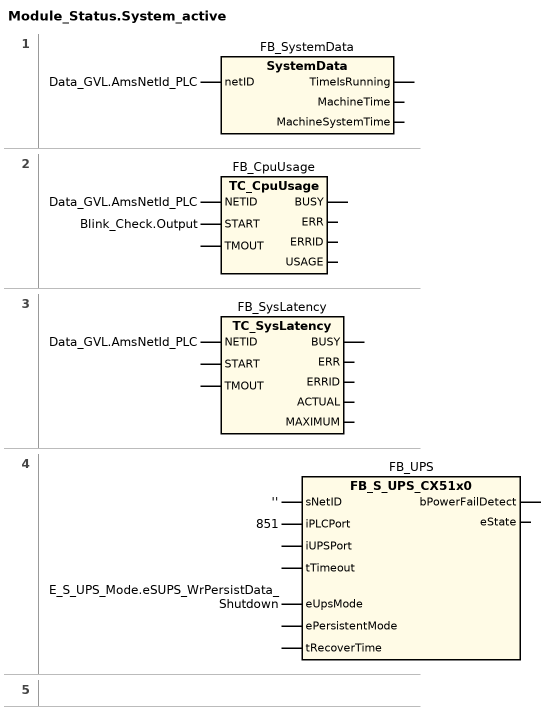
// NETWORK 1
FB_SystemData(netID := Data_GVL.AmsNetId_PLC); // SystemData

// NETWORK 2
FB_CpuUsage(NETID := Data_GVL.AmsNetId_PLC, START := Blink_Check.Output); // TC_CpuUsage

// NETWORK 3
FB_SysLatency(NETID := Data_GVL.AmsNetId_PLC); // TC_SysLatency

// NETWORK 4
FB_UPS(sNetID := '', iPLCPort := 851, eUpsMode := E_S_UPS_Mode.eSUPS_WrPersistData_Shutdown); // FB_S_UPS_CX51x0

// NETWORK 5
END_ACTION

END_PROGRAM

// ---- POUs/Function_Block/General/Ethercat_Status.TcPOU
FUNCTION_BLOCK Ethercat_Status
VAR_IN_OUT 
	stSlaveCurrentState			: stEcSlaveState;
END_VAR
VAR_INPUT
   bEnable: BOOL;                                               (*Enabling FB on rising edge*)
   sNetId: STRING;                                              (*Master's EtherCAT NetId*)
   nSlaveAddr: UINT;                                            (*Slave's EtherCAT address*)
END_VAR
VAR_OUTPUT
   bDone: BOOL;                                                 (*Successfully done*)
   iMessage: STRING (10);                                       (*String message*)
   bError: BOOL;                                                (*Error detected*)
   nErrId: UDINT;                                               (*ADS error code*)
   stActualState: ST_EcSlaveState;                              (*Actual slave status*)
END_VAR
VAR
   iStep: INT;
   fbTrigger: R_TRIG;
   fbGetSlaveState: FB_EcGetSlaveState;
   fbSetSlaveState: FB_EcSetSlaveState;
END_VAR

CASE iStep OF
   0:  (*Starting*)
       fbTrigger(CLK := bEnable);                              // Memicu fungsi fbTrigger saat sinyal bEnable aktif
          IF fbTrigger.Q THEN                                   // Jika sinyal keluaran fbTrigger aktif
             iMessage 				   		:='PROCESSING';      // Pesan status diatur menjadi 'PROCESSING'
			 stSlaveCurrentState.ERROR 		:= FALSE ;           // Status error diatur menjadi FALSE
			 stSlaveCurrentState.PROCESSING := TRUE ;            // Status proses diatur menjadi TRUE
			 stSlaveCurrentState.Init 		:= FALSE ;            // Status init diatur menjadi FALSE
			 stSlaveCurrentState.OP    		:= FALSE ;            // Status operasi diatur menjadi FALSE
             bError := FALSE;                                   // Mereset status kesalahan menjadi FALSE
             iStep := 10;                                       // Melangkah ke langkah berikutnya
          END_IF;

   10:  (*Reading slave's EtherCAT status*)
       fbGetSlaveState(                                        // Memanggil fungsi fbGetSlaveState untuk membaca status slave EtherCAT
          sNetId := sNetId,                                    // Memasukkan NetId dari slave
          nSlaveAddr := nSlaveAddr,                            // Memasukkan alamat slave
          bExecute := TRUE);                                   // Menjalankan fungsi untuk eksekusi
             IF fbGetSlaveState.bBusy THEN                     // Jika fungsi masih sibuk membaca
                iStep := 20 ;                                   // Melangkah ke langkah berikutnya
             END_IF;

   20:  (*Still reading slave's EtherCAT status*)
       fbGetSlaveState(bExecute := TRUE);                      // Melanjutkan membaca status slave EtherCAT
          IF NOT(fbGetSlaveState.bBusy) THEN                   // Jika proses membaca telah selesai
             (*Successful*)                                    // Jika berhasil
             IF NOT(fbGetSlaveState.bError) THEN               // Jika tidak ada kesalahan
                stActualState := fbGetSlaveState.state;        // Menyimpan status aktual slave yang dibaca
                fbGetSlaveState(bExecute := FALSE);            // Me-reset fungsi fbGetSlaveState
                iStep := 30;                                   // Melangkah ke langkah berikutnya
             (*Error*)                                        // Jika terjadi kesalahan
             ELSE
                iMessage						:= 'ERROR';       // Pesan status diatur menjadi 'ERROR'
				stSlaveCurrentState.ERROR 		:= TRUE;        // Status error diatur menjadi TRUE
				stSlaveCurrentState.PROCESSING  := FALSE ;     // Status proses diatur menjadi FALSE
				stSlaveCurrentState.Init 		:= FALSE ;      // Status init diatur menjadi FALSE
				stSlaveCurrentState.OP    		:= FALSE ;      // Status operasi diatur menjadi FALSE
                bError := TRUE;                                // Status kesalahan diatur menjadi TRUE
                nErrId := fbGetSlaveState.nErrId;              // Menyimpan ID kesalahan
                fbGetSlaveState(bExecute := FALSE);            // Me-reset fungsi fbGetSlaveState
                iStep := 0;                                    // Kembali ke langkah awal
             END_IF;
          END_IF;

   30:  (*Checking if slave's EtherCAT status equals 'OP'*)
       IF stActualState.deviceState = EC_DEVICE_STATE_OP THEN  // Jika status slave adalah 'OP'
          iMessage := 'OP';                                    // Pesan status diatur menjadi 'OP'
		  stSlaveCurrentState.ERROR 		:= FALSE;             // Status error diatur menjadi FALSE
		  stSlaveCurrentState.PROCESSING  	:= FALSE ;          // Status proses diatur menjadi FALSE
		  stSlaveCurrentState.Init 			:= FALSE ;          // Status init diatur menjadi FALSE
		  stSlaveCurrentState.OP    		:= TRUE ;            // Status operasi diatur menjadi TRUE
          bDone := TRUE;                                       // Operasi selesai
          iStep := 0;                                           // Kembali ke langkah awal
       ELSE                                                    // Jika status slave bukan 'OP'
          iStep := 40;                                          // Melangkah ke langkah berikutnya
       END_IF;

   
   40:  (*Setting slave into 'INIT' status*)
       fbSetSlaveState(                          // Memanggil fungsi fbSetSlaveState untuk mengatur status slave
          sNetId := sNetId,                      // Menentukan ID jaringan EtherCAT
          nSlaveAddr := nSlaveAddr,              // Menentukan alamat slave EtherCAT
          bExecute := TRUE,                      
          reqState := EC_DEVICE_STATE_INIT);     // Menentukan status yang diminta untuk diatur (INIT)
             IF fbSetSlaveState.bBusy THEN      // Jika fungsi fbSetSlaveState sedang sibuk
                iStep := 50;                    // Langkah berikutnya adalah 50
             END_IF;                            // Akhir dari kondisi IF

   50:  (*Still setting slave into 'INIT' status*)
       fbSetSlaveState(bExecute := TRUE);
          IF NOT(fbSetSlaveState.bBusy) THEN
             (*Successful*)
             IF NOT(fbSetSlaveState.bError) THEN
                fbSetSlaveState(bExecute := FALSE);             // Me-reset fungsi fbSetSlaveState
                iStep := 60;                                   // Melangkah ke langkah berikutnya
             (*Error*)
             ELSE
                iMessage 						:= 'ERROR';        // Pesan status diatur menjadi 'ERROR'
				stSlaveCurrentState.ERROR 		:= TRUE;         // Status error diatur menjadi TRUE
				stSlaveCurrentState.PROCESSING  := FALSE ;      // Status proses diatur menjadi FALSE
				stSlaveCurrentState.Init 		:= FALSE ;       // Status init diatur menjadi FALSE
				stSlaveCurrentState.OP    		:= FALSE ;       // Status operasi diatur menjadi FALSE
                bError := TRUE;                                // Status kesalahan diatur menjadi TRUE
                nErrId := fbSetSlaveState.nErrId;              // Menyimpan ID kesalahan
                fbSetSlaveState(bExecute := FALSE);            // Me-reset fungsi fbSetSlaveState
                iStep := 0;                                    // Kembali ke langkah awal
             END_IF;
          END_IF;

   60:  (*Reading slave's EtherCAT status*)
       fbGetSlaveState(
          sNetId := sNetId,
          nSlaveAddr := nSlaveAddr,
          bExecute := TRUE);
             IF fbGetSlaveState.bBusy THEN
                iStep := 70;
             END_IF;

   70:  (*Still reading slave's EtherCAT status*)
       fbGetSlaveState(bExecute := TRUE);
          IF NOT(fbGetSlaveState.bBusy) THEN
             (*Successful*)
             IF NOT(fbGetSlaveState.bError) THEN
                stActualState := fbGetSlaveState.state;         // Menyimpan status aktual slave yang dibaca
                fbGetSlaveState(bExecute := FALSE);            // Me-reset fungsi fbGetSlaveState
                iStep := 80;                                   // Melangkah ke langkah berikutnya
             (*Error*)
             ELSE
                iMessage 						:= 'ERROR';        // Pesan status diatur menjadi 'ERROR'
				stSlaveCurrentState.ERROR 		:= TRUE;         // Status error diatur menjadi TRUE
				stSlaveCurrentState.PROCESSING  := FALSE ;      // Status proses diatur menjadi FALSE
				stSlaveCurrentState.Init 		:= FALSE ;       // Status init diatur menjadi FALSE
				stSlaveCurrentState.OP    		:= FALSE ;       // Status operasi diatur menjadi FALSE
                bError := TRUE;                                // Status kesalahan diatur menjadi TRUE
                nErrId := fbGetSlaveState.nErrId;              // Menyimpan ID kesalahan
                fbGetSlaveState(bExecute := FALSE);            // Me-reset fungsi fbGetSlaveState
                iStep := 0;                                    // Kembali ke langkah awal
             END_IF;
          END_IF;

   80:  (*Checking if slave's EtherCAT status equals 'INIT'*)
       IF stActualState.deviceState = EC_DEVICE_STATE_INIT THEN // Jika status slave adalah 'INIT'
          iMessage 							:= 'INIT';         // Pesan status diatur menjadi 'INIT'
		  stSlaveCurrentState.ERROR 		:= FALSE;            // Status error diatur menjadi FALSE
		  stSlaveCurrentState.PROCESSING    := FALSE ;         // Status proses diatur menjadi FALSE
		  stSlaveCurrentState.Init 			:= TRUE ;           // Status init diatur menjadi TRUE
		  stSlaveCurrentState.OP    		:= FALSE ;          // Status operasi diatur menjadi FALSE
          iStep := 90;                                         // Melangkah ke langkah berikutnya
       ELSE                                                     // Jika status slave bukan 'INIT'
          iMessage 							:= 'ERROR';        // Pesan status diatur menjadi 'ERROR'
		  stSlaveCurrentState.ERROR 		:= TRUE;             // Status error diatur menjadi TRUE
		  stSlaveCurrentState.PROCESSING  	:= FALSE ;          // Status proses diatur menjadi FALSE
		  stSlaveCurrentState.Init 			:= FALSE ;          // Status init diatur menjadi FALSE
		  stSlaveCurrentState.OP    		:= FALSE ;          // Status operasi diatur menjadi FALSE
          bError := TRUE;                                      // Status kesalahan diatur menjadi TRUE
          iStep := 0;                                          // Kembali ke langkah awal
       END_IF;

   90:  (*Setting slave into 'OP' status*)
       fbSetSlaveState(
          sNetId := sNetId,
          nSlaveAddr := nSlaveAddr,
          bExecute := TRUE,
          reqState := EC_DEVICE_STATE_OP);
             IF fbSetSlaveState.bBusy THEN
                iStep := 100;
             END_IF;

   100: (*Still setting slave into 'OP' status*)
       fbSetSlaveState(bExecute := TRUE);
          IF NOT(fbSetSlaveState.bBusy) THEN
             (*Successful*)
             IF NOT(fbSetSlaveState.bError) THEN
                fbSetSlaveState(bExecute := FALSE);             // Me-reset fungsi fbSetSlaveState
                iStep := 110;                                  // Melangkah ke langkah berikutnya
             (*Error*)
             ELSE
                iMessage 						:= 'ERROR';        // Pesan status diatur menjadi 'ERROR'
				stSlaveCurrentState.ERROR 		:= TRUE;         // Status error diatur menjadi TRUE
				stSlaveCurrentState.PROCESSING  := FALSE ;      // Status proses diatur menjadi FALSE
				stSlaveCurrentState.Init 		:= FALSE ;       // Status init diatur menjadi FALSE
				stSlaveCurrentState.OP    		:= FALSE ;       // Status operasi diatur menjadi FALSE
                bError := TRUE;                                // Status kesalahan diatur menjadi TRUE
                nErrId := fbSetSlaveState.nErrId;              // Menyimpan ID kesalahan
                fbSetSlaveState(bExecute := FALSE);            // Me-reset fungsi fbSetSlaveState
                iStep := 0;                                    // Kembali ke langkah awal
             END_IF;
          END_IF;

   110: (*Reading slave's EtherCAT status*)
       fbGetSlaveState(
          sNetId := sNetId,
          nSlaveAddr := nSlaveAddr,
          bExecute := TRUE);
             IF fbGetSlaveState.bBusy THEN
                iStep := 120;
             END_IF;

   120: (*Still reading slave's EtherCAT status*)
       fbGetSlaveState(bExecute := TRUE);
          IF NOT(fbGetSlaveState.bBusy) THEN
             (*Successful*)
             IF NOT(fbGetSlaveState.bError) THEN
                stActualState := fbGetSlaveState.state;         // Menyimpan status aktual slave yang dibaca
                fbGetSlaveState(bExecute := FALSE);            // Me-reset fungsi fbGetSlaveState
                iStep := 130;                                  // Melangkah ke langkah berikutnya
             (*Error*)
             ELSE
                iMessage 						:= 'ERROR';        // Pesan status diatur menjadi 'ERROR'
				stSlaveCurrentState.ERROR 		:= TRUE;         // Status error diatur menjadi TRUE
				stSlaveCurrentState.PROCESSING  := FALSE ;      // Status proses diatur menjadi FALSE
				stSlaveCurrentState.Init 		:= FALSE ;       // Status init diatur menjadi FALSE
				stSlaveCurrentState.OP    		:= FALSE ;       // Status operasi diatur menjadi FALSE
                bError 							:= TRUE;        // Status kesalahan diatur menjadi TRUE
                nErrId := fbGetSlaveState.nErrId;              // Menyimpan ID kesalahan
                fbGetSlaveState(bExecute := FALSE);            // Me-reset fungsi fbGetSlaveState
                iStep := 0;                                    // Kembali ke langkah awal
             END_IF;
          END_IF;

   130: (*Checking if slave's EtherCAT status equals 'OP'*)
       IF stActualState.deviceState = EC_DEVICE_STATE_OP THEN   // Jika status slave adalah 'OP'
          iMessage 							:= 'OP';            // Pesan status diatur menjadi 'OP'
		  stSlaveCurrentState.ERROR 		:= FALSE;             // Status error diatur menjadi FALSE
		  stSlaveCurrentState.PROCESSING  	:= FALSE ;          // Status proses diatur menjadi FALSE
		  stSlaveCurrentState.Init 			:= FALSE ;          // Status init diatur menjadi FALSE
		  stSlaveCurrentState.OP    		:= TRUE ;            // Status operasi diatur menjadi TRUE
          iStep := 140;                                        // Melangkah ke langkah berikutnya
       ELSE                                                     // Jika status slave bukan 'OP'
          iMessage := 'ERROR';                                 // Pesan status diatur menjadi 'ERROR'
		  stSlaveCurrentState.ERROR 		:= TRUE;             // Status error diatur menjadi TRUE
	      stSlaveCurrentState.PROCESSING 	:= FALSE ;          // Status proses diatur menjadi FALSE
	      stSlaveCurrentState.Init 			:= FALSE ;          // Status init diatur menjadi FALSE
		  stSlaveCurrentState.OP    		:= FALSE ;          // Status operasi diatur menjadi FALSE
          bError := TRUE;                                      // Status kesalahan diatur menjadi TRUE
          iStep := 0;                                          // Kembali ke langkah awal
       END_IF;

   140: (*Setting 'OP' status successfully done*)
       bDone := TRUE;                                          // Operasi selesai
       iStep := 0;                                             // Kembali ke langkah awal
END_CASE;

END_FUNCTION_BLOCK

// ---- POUs/Function_Block/General/SystemData.TcPOU
FUNCTION_BLOCK SystemData
VAR_INPUT
	netID: T_AmsNetID;
END_VAR
VAR_OUTPUT
	TimeIsRunning: BOOL;
	
	MachineTime: DT;
	MachineSystemTime: TIMESTRUCT;
END_VAR
VAR
	GetTime: NT_GetTime;
	synchTime: TON;
	
	F_Trig_RTC: F_Trig;
	DataRTC: RTC;
END_VAR

VAR CONSTANT
	TimerCheck: TIME := T#2s;
END_VAR

synchTime(IN := NOT synchTime.Q, PT := TimerCheck); // TON
GetTime(NETID := netID, START := synchTime.Q, TMOUT := TimerCheck); // NT_GetTime
F_Trig_RTC(CLK := GetTime.BUSY AND NOT GetTime.ERR); // F_Trig
DataRTC(EN := F_Trig_RTC.Q, PDT := SYSTEMTIME_TO_DT(TIMESTR := GetTime.TIMESTR)); // RTC
TimeIsRunning S= DataRTC.Q;
MachineTime := DataRTC.CDT;
MachineSystemTime := DT_TO_SystemTime(dtIn := DataRTC.CDT);

END_FUNCTION_BLOCK

// ---- POUs/Function_Block/Placing/FB_CustomOffset.TcPOU
FUNCTION_BLOCK FB_CustomOffset
VAR_INPUT
	Dt_OffsetPlacing	: stCustomOffset;
	iCounter			: INT;
END_VAR
VAR_OUTPUT
	iOffset_X			: UINT;
	iOffset_Y			: UINT;
	iLayer				: INT;
	iCycle				: INT;
END_VAR
VAR
	
END_VAR

iCycle := iCounter MOD 18;
IF iCycle=0 THEN
	iCycle:=18;
END_IF

iLayer := 1+((iCounter-1)/9);

iOffset_X := INT_TO_UINT(Dt_OffsetPlacing.iOffset_X[iCycle]);
iOffset_Y := INT_TO_UINT(Dt_OffsetPlacing.iOffset_Y[iCycle]);

END_FUNCTION_BLOCK

// ---- GlobalTextList.TcGTLO
TEXTLIST GlobalTextList
  1836 = ' '
  4414 = '%3.1f'
  100 = '%3.1f %'
  2062 = '%3.3f'
  4760 = '%3.3f %'
  950 = '%3.5f'
  2819 = '%3.5f %'
  989 = '%5.1f hour'
  2126 = '%5.2f'
  1746 = '%5.2f %'
  314 = '%5.2f%'
  430 = '%5.3f H'
  4455 = '%5.3f hour'
  2043 = '%5.3f hours'
  0 = '%5.3f our'
  1761 = '%5.4 ms'
  1143 = '%5.4f H'
  3371 = '%i'
  1125 = '%I'
  2829 = '%i  ms'
  169 = '%i %'
  818 = '%i ms'
  1785 = '%s'
  1019 = '%S'
  9 = '1'
  1280 = '10'
  4636 = '1000'
  1709 = '1000\tPush\xa0Button\xa0Run\xa0at P2\n1001\tPush\xa0Button\xa0Stop\xa0at P2\n1002\tPush\xa0Button\xa0Alarm\xa0Reset\xa0at\xa0P2\n1003\tPush Button Acknowledge at P2\n1004\tAuto/Manual Switch (0=Running Mode, 1=Test Mode)\n1005\tEmergency\xa0Stop\xa0at\xa0P2\n1006\t\n1007\tPSR Back at Loaded Pallet Outfeed Roller Conveyor 5\n1008\tPSR Front at Loaded Pallet Outfeed Roller Conveyor 5\n1009\tSafety Light Curtain\n1010\t\n1011\t\n1012\t\n1013\tPSR Back at Detect Loaded Pallet Buffer Roller Conv 2 \n1014\tPSR Front at Detect Loaded Pallet Buffer Roller Conv 2 \n1015\tFeedback Loaded Pallet Outfeed Roller Conveyor 5 is Running'
  3712 = '1000\tPush\xa0Button\xa0Run\xa0at P2\n1001\tPush\xa0Button\xa0Stop\xa0at P2\n1002\tPush\xa0Button\xa0Alarm\xa0Reset\xa0at\xa0P2\n1003\tPush Button Acknowledge at P2\n1004\tAuto/Manual Switch (0=Running Mode, 1=Test Mode)\n1005\tEmergency\xa0Stop\xa0at\xa0P2\n1006\t\n1007\tPSR Back at Loaded Pallet Outfeed Roller Conveyor 5 (GL6-P4212)\n1008\tPSR Front at Loaded Pallet Outfeed Roller Conveyor 5 (GL6-P4212)\n1009\tSafety Light Curtain\n1010\t\n1011\t\n1012\t\n1013\tPSR Back at Detect Loaded Pallet Buffer Roller Conv 2 (GL6-P4212)\n1014\tPSR Front at Detect Loaded Pallet Buffer Roller Conv 2 (GL6-P4212)\n1015\tFeedback Loaded Pallet Outfeed Roller Conveyor 5 is Running'
  5284 = '1000\tPush\xa0Button\xa0Run\xa0at\xa0Main Panel\n1001\tPush\xa0Button\xa0Stop\xa0at\xa0Main Panel\n1002\tPush\xa0Button\xa0Alarm\xa0Reset\xa0at\xa0Main Panel\n1003\tPush Button Acknowledge at Main Panel\n1004\tEmergency\xa0Stop\xa0at\xa0Infeed Panel\n1005\tAuto/Manual Switch (0=Running Mode, 1=Test Mode)\n1006\t\n1007\t\n1008\t\n1009\t\n1010\t\n1011\t\n1012\t\n1013\t\n1014\t\n1015\tPressure Switch for Main Panel\n'
  759 = '1000 - Push\xa0Button\xa0Run\xa0at P2'
  428 = '1001 - Push\xa0Button\xa0Stop\xa0at P2\n'
  429 = '1002 - Push\xa0Button\xa0Alarm\xa0Reset\xa0at\xa0P2\n'
  181 = '1003 - Push Button Acknowledge at P2'
  739 = '1004 - Auto/Manual Switch'
  348 = '1005 - Emergency\xa0Stop\xa0at\xa0P2'
  910 = '1006\n'
  720 = '1007 - Feedback Buffer Roller 2  Conveyor is Running'
  371 = '1007 - PSR Back at Detect Loaded Pallet Buffer Roller Conv 2 (GL6-P4212)'
  19 = '1008 - Feedback Loaded Pallet Buffer Conveyor 1 is Running'
  1082 = '1008 - PSR Front at Detect Loaded Pallet Buffer Roller Conv 2 (GL6-P4212)'
  879 = '1009 - Safety Light Curtain\n'
  1148 = '1010 - Safety Door Solenoid Channel 1'
  877 = '1011 - Safety Door Solenoid Channel 2'
  1006 = '1012 '
  486 = '1013 - PSR Back at Loaded Pallet Outfeed Roller Conveyor 5 (GL6-P4212)'
  426 = '1014 - PSR Front at Loaded Pallet Outfeed Roller Conveyor 5 (GL6-P4212)'
  889 = '1015 - Feedback Loaded Pallet Outfeed Roller Conveyor 5 is Running'
  1164 = '10xx'
  1517 = '11'
  3803 = '1100\tFeedback Box Transfer Modullar Conveyor 1 is Running\n1101\tFeedback Box Transfer Modullar Conveyor 2 is Running\n1102\tFeedback Box Transfer Modullar Conveyor 3 is Running\n1103\tFeedback Box Transfer Modullar Conveyor 4 is Running\n1104\tFeedback Box Infeed Roller Conveyor is Running\n1105\tFeedback Box Stop & Go Conveyor is Running\n1106\tFeedback Buffer Roller 1  Conveyor is Running\n1107\tFeedback Buffer Roller 2  Conveyor is Running\n1108\tFeedback Loaded Pallet Buffer Conveyor 1 is Running\n1109\tFeedback Loaded Pallet Outfeed Roller Conveyor 1 is Running\n1110\tFeedback Right Angel is Running\n1111\tFeedback Right Angel Lifter is Running\n1112\tFeedback Loaded Pallet Outfeed Roller Conveyor 2 is Running\n1113\tFeedback Loaded Pallet Outfeed Roller Conveyor 3 is Running\n1114\tFeedback Loaded Pallet Outfeed Roller Conveyor 4 is Running\n1115\tFeedback Loaded Pallet Buffer 2 is Running'
  1220 = '1100\tFeedback Box Transfer Modullar Conveyor 1 is Running\n1101\tFeedback Box Transfer Modullar Conveyor 2 is Running\n1102\tFeedback Box Transfer Modullar Conveyor 3 is Running\n1103\tFeedback Box Transfer Modullar Conveyor 4 is Running\n1104\tFeedback Box Infeed Roller Conveyor is Running\n1105\tFeedback Box Stop & Go Conveyor is Running\n1106\tFeedback Buffer Roller 1  Conveyor is Running\n1107\tFeedback Buffer Roller 2  Conveyor is Running\n1108\tFeedback Loaded Pallet Buffer Conveyor 1 is Running\n1109\tFeedback Loaded Pallet Outfeed Roller Conveyor 1 is Running\n1110\tFeedback Right Angel is Running\n1111\tFeedback Right Angel Lifter is Running\n1112\tFeedback Loaded Pallet Outfeed Roller Conveyor 2 is Running\n1113\tFeedback Loaded Pallet Outfeed Roller Conveyor 3 is Running\n1114\tFeedback Loaded Pallet Outfeed Roller Conveyor 4 is Running\n1115\tFeedback Loaded Pallet Buffer 2 is Running (Take Over Motor Lama)'
  235 = '1100 - Feedback Box Transfer Modullar Conveyor 1 is Running'
  1130 = '1101 - Feedback Box Transfer Modullar Conveyor 2 is Running\n'
  266 = '1102 - Feedback Box Transfer Modullar Conveyor 3 is Running'
  523 = '1103 - Feedback Box Transfer Modullar Conveyor 4 is Running'
  310 = '1104 - Feedback Box Infeed Roller Conveyor is Running'
  352 = '1105 - Feedback Box Stop & Go Conveyor is Running'
  885 = '1106 - Feedback Buffer Roller 1  Conveyor is Running'
  295 = '1109 - Feedback Loaded Pallet Outfeed Roller Conveyor 1 is Running'
  857 = '1110 - Feedback Right Angel is Running'
  142 = '1111 - Feedback Right Angel Lifter is Running'
  477 = '1112 - Feedback Loaded Pallet Outfeed Roller Conveyor 2 is Running'
  856 = '1113 - Feedback Loaded Pallet Outfeed Roller Conveyor 3 is Running'
  17 = '1114 - Feedback Loaded Pallet Outfeed Roller Conveyor 4 is Running'
  1256 = '1115 - Feedback Loaded Pallet Buffer 2 is Running'
  701 = '11xx'
  653 = '12'
  728 = '1200'
  3570 = '1200\t\n1201\t\n1202\t\n1203\t\n1204\tPSR Back at Detect Loaded Pallet Buffer Roller Conv 1\n1205\tPSR Front at Detect Loaded Pallet Buffer Roller Conv 1\n1206\tPSR Back at Loaded Pallet Outfeed Roller Conveyor 1\n1207\tPSR Front at Loaded Pallet Outfeed Roller Conveyor 1\n1208\tPSR Back at Loaded Pallet Outfeed Roller Conveyor 2\n1209\tPSR Front at Loaded Pallet Outfeed Roller Conveyor 2\n1210\tProximity Sensor at Bottom Position Pallet RA Lifter \n1211\tProximity Sensor at Top Position Pallet RA Lifter\n1212\tPSR Back at Loaded Pallet Outfeed Roller Conveyor 3 \n1213\tPSR Front at Loaded Pallet Outfeed Roller Conveyor 3 \n1214\tPSR Back at Loaded Pallet Outfeed Roller Conveyor 4 \n1215\tPSR Front at Loaded Pallet Outfeed Roller Conveyor 4'
  5027 = '1200\t\n1201\t\n1202\t\n1203\t\n1204\tPSR Back at Detect Loaded Pallet Buffer Roller Conv 1 (GL6-P4212)\n1205\tPSR Front at Detect Loaded Pallet Buffer Roller Conv 1 (GL6-P4212)\n1206\tPSR Back at Loaded Pallet Outfeed Roller Conveyor 1 (GL6-P4212)\n1207\tPSR Front at Loaded Pallet Outfeed Roller Conveyor 1 (GL6-P4212)\n1208\tPSR Back at Loaded Pallet Outfeed Roller Conveyor 2 (GL6-P4212)\n1209\tPSR Front at Loaded Pallet Outfeed Roller Conveyor 2 (GL6-P4212)\n1210\tProximity Sensor at Bottom Position Pallet RA Lifter  (E2B-M12KN08-M1-B1)\n1211\tProximity Sensor at Top Position Pallet RA Lifter (E2B-M12KN08-M1-B1)\n1212\tPSR Back at Loaded Pallet Outfeed Roller Conveyor 3 (GL6-P4212)\n1213\tPSR Front at Loaded Pallet Outfeed Roller Conveyor 3 (GL6-P4212)\n1214\tPSR Back at Loaded Pallet Outfeed Roller Conveyor 4 (GL6-P4212)\n1215\tPSR Front at Loaded Pallet Outfeed Roller Conveyor 4 (GL6-P4212)'
  4020 = '1200\t\n1201\t\n1202\t\n1203\tPSR to Check Box at Loaded Pallet Buffer Roller Conv 1\n1204\tPSR Back at Detect Loaded Pallet Buffer Roller Conv 1\n1205\tPSR Front at Detect Loaded Pallet Buffer Roller Conv 1\n1206\tPSR Back at Loaded Pallet Outfeed Roller Conveyor 1\n1207\tPSR Front at Loaded Pallet Outfeed Roller Conveyor 1\n1208\tPSR Back at Loaded Pallet Outfeed Roller Conveyor 2\n1209\tPSR Front at Loaded Pallet Outfeed Roller Conveyor 2\n1210\tProximity Sensor at Bottom Position Pallet RA Lifter \n1211\tProximity Sensor at Top Position Pallet RA Lifter\n1212\tPSR Back at Loaded Pallet Outfeed Roller Conveyor 3 \n1213\tPSR Front at Loaded Pallet Outfeed Roller Conveyor 3 \n1214\tPSR Back at Loaded Pallet Outfeed Roller Conveyor 4 \n1215\tPSR Front at Loaded Pallet Outfeed Roller Conveyor 4'
  5286 = '1200\tFeedback Box Picking roller Conveyor is Running\n1201\t\n1202\tFeedback Box Placing at Pallet Roller Conveyor 1 is Running\n1203\tFeedback Box Placing at Pallet Roller Conveyor 2 is Running\n1204\tFeedback Box Placing at Pallet Roller Conveyor 3 is Running\n1205\tFeedback Box Placing at Pallet Roller Conveyor 4  isRunning\n1206\t\n1207\t\n1208\t\n1209\t\n1210\t\n1211\tRSW Pneumatic Box Centring When Rtc\n1212\tRSW Pneumatic Gap Maker When Adv\n1213\tRSW Pneumatic Gap Maker When Rtc\n1214\tRSW Pneumatic Stopper  Transfer When Rtc\n1215\t\n'
  1003 = '1201 - Feedback Loaded Pallet Buffer 3 is Running'
  633 = '1202 - PSR Back at Detect Loaded Pallet Buffer Roller Conv (GL6-P4212)'
  3 = '1203 - PSR Front at Detect Loaded Pallet Buffer Roller Conv (GL6-P4212)'
  677 = '1204 - PSR Front at Detect Loaded Pallet Buffer Roller Conv (GL6-P4212)'
  1371 = '1205 - PSR Front at Loaded Pallet Outfeed Roller Conveyor 1 (GL6-P4212)'
  1144 = '1206 - PSR Back to Check Pallet RA Transfer Chain (GL6-P4212)'
  129 = '1207 - PSR Front to Check Pallet RA Transfer Chain (GL6-P4212)'
  2194 = '1208 - PSR Back at Loaded Pallet Outfeed Roller Conveyor 2 (GL6-P4212)'
  1414 = '1209 - PSR Front at Loaded Pallet Outfeed Roller Conveyor 2 (GL6-P4212)'
  2074 = '1210 - Proximity Sensor at Bottom Position Pallet RA Lifter  (E2B-M12KN08-M1-B1)'
  1277 = '1211 - Proximity Sensor at Top Position Pallet RA Lifter (E2B-M12KN08-M1-B1)'
  1556 = '1212 - PSR Back at Loaded Pallet Outfeed Roller Conveyor 3 (GL6-P4212)'
  1416 = '1213 - PSR Front at Loaded Pallet Outfeed Roller Conveyor 3 (GL6-P4212)'
  151 = '1214 - PSR Back at Loaded Pallet Outfeed Roller Conveyor 4 (GL6-P4212)'
  320 = '1215 - PSR Front at Loaded Pallet Outfeed Roller Conveyor 4 (GL6-P4212)'
  2569 = '12xx'
  318 = '13'
  4082 = '1300\tFeedback Automatic Pallet Dispenser is Running\n1301\tPSR Back to Check Pallet at Automatic Pallet Dispenser \n1302\tPSR Front to Check Pallet at Automatic Pallet Dispenser\n1303\tPSR to Check Stock Pallet at Automatic Pallet Dispenser\n1304\tRSW for Check Position Right Pneumatic Horizontal when Retract\n1305\tRSW for Check Position Right Pneumatic Horizontal when Advanced\n1306\tRSW for Check Position Left Pneumatic Horizontal when Retract\n1307\tRSW for Check Position Left Pneumatic Horizontal when Advanced\n1308\tPSR Transfer to Check Pallet at Automatic Pallet Dispenser \n1309\tProximity Sensor at Retract Position Right Pneumatic Vertical\n1310\tProximity Sensor at Middle Position Right Pneumatic Vertical\n1311\tProximity Sensor at Advanced Position Right Pneumatic Vertical\n1312\tProximity Sensor at  Retract Position Left Pneumatic Vertical\n1313\tProximity Sensor at Middle Position Left Pneumatic Vertical\n1314\tProximity Sensor at Advanced Position Left Pneumatic Vertical\n1315\tRequest Release Solenoid Door Outfeed'
  2849 = '1300\tFeedback Automatic Pallet Dispenser is Running\n1301\tPSR Back to Check Pallet at Automatic Pallet Dispenser (GL6-P4212)\n1302\tPSR Front to Check Pallet at Automatic Pallet Dispenser (GL6-P4212)\n1303\tPSR to Check Stock Pallet at Automatic Pallet Dispenser (GL6-P4212)\n1304\tRSW for Check Position Right Pneumatic Horizontal when Retract\n1305\tRSW for Check Position Right Pneumatic Horizontal when Advanced\n1306\tRSW for Check Position Left Pneumatic Horizontal when Retract\n1307\tRSW for Check Position Left Pneumatic Horizontal when Advanced\n1308\tPSR Transfer to Check Pallet at Automatic Pallet Dispenser (GL6-P4212)\n1309\tProximity Sensor at Retract Position Right Pneumatic Vertical\n1310\tProximity Sensor at Middle Position Right Pneumatic Vertical\n1311\tProximity Sensor at Advanced Position Right Pneumatic Vertical\n1312\tProximity Sensor at  Retract Position Left Pneumatic Vertical\n1313\tProximity Sensor at Middle Position Left Pneumatic Vertical\n1314\tProximity Sensor at Advanced Position Left Pneumatic Vertical\n1315\tRequest Release Solenoid Door Outfeed'
  4248 = '1300\tFeedback Automatic Pallet Dispenser is Running\n1301\tPSR Back to Check Pallet at Automatic Pallet Dispenser (GL6-P4212)\n1302\tPSR Front to Check Pallet at Automatic Pallet Dispenser (GL6-P4212)\n1303\tPSR to Check Stock Pallet at Automatic Pallet Dispenser (GL6-P4212)\n1304\tRSW for Check Position Right Pneumatic Horizontal when Retract\n1305\tRSW for Check Position Right Pneumatic Horizontal when Advanced\n1306\tRSW for Check Position Left Pneumatic Horizontal when Retract\n1307\tRSW for Check Position Left Pneumatic Horizontal when Advanced\n1308\tPSR Transfer to Check Pallet at Automatic Pallet Dispenser (GL6-P4212)\n1309\tProximity Sensor at Retract Position Right Pneumatic Vertical\n1310\tProximity Sensor at Middle Position Right Pneumatic Vertical\n1311\tProximity Sensor at Advanced Position Right Pneumatic Vertical (E2B-M12KN08-M1-B1)\n1312\tProximity Sensor at  Retract Position Left Pneumatic Vertical (E2B-M12KN08-M1-B1)\n1313\tProximity Sensor at Middle Position Left Pneumatic Vertical (E2B-M12KN08-M1-B1)\n1314\tProximity Sensor at Advanced Position Left Pneumatic Vertical (E2B-M12KN08-M1-B1)\n1315\tRequest Release Solenoid Door Outfeed'
  760 = '1300\tFeedback Automatic Pallet Dispenser is Running\n1301\tPSR Back to Check Pallet at Automatic Pallet Dispenser (GL6-P4212)\n1302\tPSR Front to Check Pallet at Automatic Pallet Dispenser (GL6-P4212)\n1303\tPSR to Check Stock Pallet at Automatic Pallet Dispenser (GL6-P4212)\n1304\tRSW for Check Position Right Pneumatic Horizontal when Retract\n1305\tRSW for Check Position Right Pneumatic Horizontal when Advanced\n1306\tRSW for Check Position Left Pneumatic Horizontal when Retract\n1307\tRSW for Check Position Left Pneumatic Horizontal when Advanced\n1308\tPSR Transfer to Check Pallet at Automatic Pallet Dispenser (GL6-P4212)\n1309\tProximity Sensor at Retract Position Right Pneumatic Vertical\n1310\tProximity Sensor at Middle Position Right Pneumatic Vertical (E2B-M12KN08-M1-B1)\n1311\tProximity Sensor at Advanced Position Right Pneumatic Vertical (E2B-M12KN08-M1-B1)\n1312\tProximity Sensor at  Retract Position Left Pneumatic Vertical (E2B-M12KN08-M1-B1)\n1313\tProximity Sensor at Middle Position Left Pneumatic Vertical (E2B-M12KN08-M1-B1)\n1314\tProximity Sensor at Advanced Position Left Pneumatic Vertical (E2B-M12KN08-M1-B1)\n1315\tRequest Release Solenoid Door Outfeed'
  4383 = '1300\tFeedback Automatic Pallet Dispenser is Running\n1301\tPSR Back to Check Pallet at Automatic Pallet Dispenser (GL6-P4212)\n1302\tPSR Front to Check Pallet at Automatic Pallet Dispenser (GL6-P4212)\n1303\tPSR to Check Stock Pallet at Automatic Pallet Dispenser (GL6-P4212)\n1304\tRSW for Check Position Right Pneumatic Horizontal when Retract\n1305\tRSW for Check Position Right Pneumatic Horizontal when Advanced\n1306\tRSW for Check Position Left Pneumatic Horizontal when Retract\n1307\tRSW for Check Position Left Pneumatic Horizontal when Advanced\n1308\tPSR Transfer to Check Pallet at Automatic Pallet Dispenser (GL6-P4212)\n1309\tProximity Sensor at Retract Position Right Pneumatic Vertical (E2B-M12KN08-M1-B1)\n1310\tProximity Sensor at Middle Position Right Pneumatic Vertical (E2B-M12KN08-M1-B1)\n1311\tProximity Sensor at Advanced Position Right Pneumatic Vertical (E2B-M12KN08-M1-B1)\n1312\tProximity Sensor at  Retract Position Left Pneumatic Vertical (E2B-M12KN08-M1-B1)\n1313\tProximity Sensor at Middle Position Left Pneumatic Vertical (E2B-M12KN08-M1-B1)\n1314\tProximity Sensor at Advanced Position Left Pneumatic Vertical (E2B-M12KN08-M1-B1)\n1315\tRequest Release Solenoid Door Outfeed'
  1140 = '1300 - PSR to Detect Infeed Box Roller Conv. (GTE6-P4212)'
  312 = '1301 - PSR Back to Detect Box at Stop & Go Conv. (GL6-P4212)'
  73 = '1302 - PSR Front to Detect Box at Stop & Go Conv. (GTE6-P4212)\n'
  18 = '1303 - PSR to Detect Stopper 1 Conv. (GL6-P4212)'
  268 = '1304 - PSR to Detect Stopper 2 Conv. (GL6-P4212)'
  1076 = '1305'
  480 = '1306 - PSR Front to Detect Puhser for Buffer Roller 1. (GTE6-P4212)'
  1312 = '1307 - PSR Back to Detect Puhser for Buffer Roller 1. (GTE6-P4212)'
  99 = '1308 - PSR Front to Detect Puhser for Buffer Roller 2. (GTE6-P4212)'
  1334 = '1309 - PSR Middle to Detect for Buffer Roller 2. (GL6-P4212)'
  1065 = '1310 - PSR Back to Detect Puhser for Buffer Roller 2. (GTE6-P4212)'
  936 = '1311'
  812 = '1312 - PSR Front at Transfer Modular Conv 1 (GL6-P4212)'
  1078 = '1313 - PSR Front at Transfer Modular Conv 2 (GL6-P4212)'
  1372 = '1314 - PSR Back at Transfer Modular  Conv 2 (GL6-P4212)'
  926 = '1315 - PSR Front at Transfer Modular Conv 3 (GL6-P4212)'
  4150 = '13xx'
  333 = '14'
  525 = '1400'
  155 = '1400\tPSR 4 to Detect Box at Picking Conv.  (GTE6-P4212)\n1401\t\n1402\t\n1403\t\n1404\t\n1405\tPSR 1 to Detect Box at Picking Conv.  (GTE6-P4212)\n1406\tPSR 2 to Detect Box at Picking Conv. (GTE6-P4212)\n1407\tPSR 3 to Detect Box at Picking Conv.  (GTE6-P4212)\n1408\tPSR Front to Detect for Empty Transfer Infeed Roller. (GL6-P4212)\n1409\tPSR Middle to Detect for Empty Transfer Infeed Roller. (GL6-P4212)\n1410\tPSR Back to Detect for Empty Transfer Infeed Roller. (GL6-P4212)\n1411\t\n1412\t\n1413\t\n1414\tRequest Release Solenoid Door Robot\n1415\tFeedback Relay Solenoid Door Robot\n'
  3412 = '1400\tRequest Release Solenoid Door Wrapper\n1401\tRSW Pneumatic Stopper 1 When Rtc\n1402\tRSW Pneumatic Stopper 2 When Rtc\n1403\tRSW Pneumatic Pusher Stop&Go  Adv\n1404\tRSW Pneumatic Pusher Stop&Go  Rtc\n1405\tRSW Pneumatic Pusher Buffer Roller 1 Adv\n1406\tRSW Pneumatic Pusher Buffer Roller  1 Rtc\n1407\tRSW Pneumatic Pusher Buffer Roller  2 Adv\n1408\tRSW Pneumatic Pusher Buffer Roller  2 Rtc\n1409\tFeedback Relay Solenoid Door 1 (Outfeed)\n1410\tFeedback Relay Solenoid Door 2 (Wrapper)\n1411\t\n1412\t\n1413\t\n1414\tInterlock Feedback Pallet Ready at Infeed Dispenser\n1415\tInterlock Feedback Pallet Ready at Unloading'
  3015 = '1400\tRequest Release Solenoid Door Wrapper\n1401\tRSW Pneumatic Stopper 1 When Rtc\n1402\tRSW Pneumatic Stopper 2 When Rtc\n1403\tRSW Pneumatic Pusher Stop&Go  Adv\n1404\tRSW Pneumatic Pusher Stop&Go  Rtc\n1405\tRSW Pneumatic Pusher Buffer Roller 1 Adv\n1406\tRSW Pneumatic Pusher Buffer Roller  1 Rtc\n1407\tRSW Pneumatic Pusher Buffer Roller  2 Adv\n1408\tRSW Pneumatic Pusher Buffer Roller  2 Rtc\n1409\tFeedback Relay Solenoid Door 1 (Outfeed)\n1410\tFeedback Relay Solenoid Door 2 (Wrapper)\n1411\tRSW Pneumatic Stopper Modullar When Adv\n1412\tRSW Pneumatic Stopper Modullar When Rtc\n1413\t\n1414\tInterlock Feedback Pallet Ready at Infeed Dispenser\n1415\tInterlock Feedback Pallet Ready at Unloading'
  1373 = '1401 - RSW Pneumatic Stopper 1 When Rtc'
  1546 = '1402 - RSW Pneumatic Stopper 2 When Rtc\n'
  1389 = '1403 - RSW Pneumatic Pusher Stop&Go  Adv'
  548 = '1404 - RSW Pneumatic Pusher Stop&Go  Rtc'
  749 = '1405 - RSW Pneumatic Pusher Buffer Roller 1 Adv'
  413 = '1406 - RSW Pneumatic Pusher Buffer Roller  1 Rtc'
  672 = '1407 - RSW Pneumatic Pusher Buffer Roller  2 Adv'
  1618 = '1408 - RSW Pneumatic Pusher Buffer Roller  2 Rtc'
  1811 = '1409\n'
  128 = '1410'
  1613 = '1411 - Feedback Relay Solenoid Door Coil Channel 1'
  1087 = '1412 - Feedback Relay Solenoid Door Coil Channel 2'
  786 = '1413 - EDM for STO Solenoid Door Coil'
  1752 = '1414 - Interlock Status Running Outfeed Existing'
  51 = '1415 - Interlock Feedback Pallet Ready Conveyor Existing'
  1096 = '14xx'
  2435 = '15'
  1353 = '1500\tPSR Back at Placing Conv 1 (GL6-P4212)\n1501\tPSR Middle at Placing Conv 1 (GL6-P4212)\n1502\tPSR Front at Placing Conv 1 (GL6-P4212)\n1503\tPSR Back at Placing Conv 2 (GL6-P4212)\n1504\tPSR Front at Placing Conv 2 (GL6-P4212)\n1505\tPSR Back at Placing Conv 3 (GL6-P4212)\n1506\tPSR Front at Placing Conv 3 (GL6-P4212)\n1507\tPSR Back at Placing Conv 4 (GL6-P4212)\n1508\tPSR Middle at Placing Conv 4 (GL6-P4212)\n1509\tPSR Front at Placing Conv 4 (GL6-P4212)\n1510\t\n1511\t\n1512\t\n1513\t\n1514\t\n1515\t'
  575 = '1500\tPush\xa0Button\xa0Run\xa0at\xa0Dispenser\n1501\tPush\xa0Button\xa0Stop\xa0at\xa0Dispenser\n1502\tPush\xa0Button\xa0Alarm\xa0Reset\xa0at\xa0Dispenser\n1503\tPush Button Acknowledge at Dispenser\n1504\tAuto/Manual Switch (0=Running Mode, 1=Test Mode) at Dispenser\n1505\tEmergency\xa0Stop\xa0at\xa0Dispenser\n1506\tManual Switch for Test Pneumatic Vertical UP\n1507\tManual Switch for Test Pneumatic Vertical DOWN\n1508\tManual Switch for Test Pneumatic Horizontal\n1509\tManual Switch for Test Motor Automatic Pallet Roller Conv.\n1510\tWrapper Ready to Receive\n1511\tEnd of Transfer Pallet in Infeed\n1512\tPallet Ready in Outfeed\n1513\tEmergency Stop Wrapper is Active\n1514\tStatus Bypass Wrapper Existing\n1515\tPressure Switch for Pallet Dispenser'
  4440 = '15xx'
  659 = '16'
  1394 = '1600\tPSR to Detect Infeed Box Roller Conv.\n1601\tPSR Back to Detect Pusher for Stop & Go Conv. \n1602\tPSR Front to Detect Box at Stop & Go Conv. \n1603\tPSR to Detect Stopper 1 Conv. \n1604\tPSR to Detect Stopper 2 Conv.\n1605\t\n1606\tPSR Back to Detect Box at Buffer Roller 1.\n1607\tPSR Front to Detect Pusher for Buffer Roller 1.\n1608\tPSR Back to Detect Box at Buffer Roller 2. \n1609\tPSR Middle to Detect Box at Buffer Roller 2.\n1610\tPSR Front to Detect Puhser for Buffer Roller 2. \n1611\t\n1612\tPSR Front at Transfer Modular Conv 1\n1613\tPSR Back at Transfer Modular Conv 1\n1614\tPSR Front at Transfer Modular Conv 2\n1615\tPSR Front at Transfer Modular Conv 3'
  3893 = '1600\tPSR to Detect Infeed Box Roller Conv.\n1601\tPSR Back to Detect Pusher for Stop & Go Conv. \n1602\tPSR Front to Detect Box at Stop & Go Conv. \n1603\tPSR to Detect Stopper 1 Conv. \n1604\tPSR to Detect Stopper 2 Conv.\n1605\t\n1606\tPSR Back to Detect Box at Buffer Roller 1.\n1607\tPSR Front to Detect Pusher for Buffer Roller 1.\n1608\tPSR Back to Detect Box at Buffer Roller 2. \n1609\tPSR Middle to Detect Box at Buffer Roller 2.\n1610\tPSR Front to Detect Puhser for Buffer Roller 2. \n1611\tPSR Front at Transfer Modular Conv 4\n1612\tPSR Front at Transfer Modular Conv 2\n1613\tPSR Back at Transfer Modular Conv 3\n1614\tPSR Front at Transfer Modular Conv 3\n1615\tPSR Back at Transfer Modular Conv 4\n'
  5306 = '1600\tPSR to Detect Infeed Box Roller Conv. (GTE6-P4212)\n1601\tPSR Back to Detect Pusher for Stop & Go Conv. (GTE6-P4212)\n1602\tPSR Front to Detect Box at Stop & Go Conv. (GTE6-P4212)\n1603\tPSR to Detect Stopper 1 Conv. (GL6-P4212)\n1604\tPSR to Detect Stopper 2 Conv. (GL6-P4212)\n1605\t\n1606\tPSR Back to Detect Box at Buffer Roller 1. (GTE6-P4212)\n1607\tPSR Front to Detect Pusher for Buffer Roller 1. (GTE6-P4212)\n1608\tPSR Back to Detect Box at Buffer Roller 2. (GTE6-P4212)\n1609\tPSR Middle to Detect Box at Buffer Roller 2. (GL6-P4212)\n1610\tPSR Front to Detect Puhser for Buffer Roller 2. (GTE6-P4212)\n1611\t\n1612\tPSR Front at Transfer Modular Conv 1 (GL6-P4212)\n1613\tPSR Back at Transfer Modular Conv 1 (GL6-P4212)\n1614\tPSR Front at Transfer Modular Conv 2 (GL6-P4212)\n1615\tPSR Front at Transfer Modular Conv 3 (GL6-P4212)'
  4409 = '16xx'
  1007 = '17'
  2068 = '18'
  440 = '19'
  2344 = '2'
  2645 = '20'
  3495 = '2000\tIndicator\xa0Machine\xa0Running\xa0at\xa0Main Panel\n2001\tIndicator\xa0Machine\xa0Error\xa0at\xa0Main Panel\n2002\tIndicator Tower\xa0Lamp\xa0Red\n2003\tIndicator Tower\xa0Lamp\xa0Yellow\n2004\tIndicator Tower\xa0Lamp\xa0Green\n2005\tIndicator Tower\xa0Lamp\xa0Blue\n2006\tIndicator Buzzer\n2007\tIndicator Acknowledge at Main Panel\n2008\tIndicator Auto Mode Main Panel\n2009\tIndicator Manual Mode Main Panel\n2010\t\n2011\t\n2012\t\n2013\t\n2014\t\n2015\t'
  119 = '2000\tIndicator\xa0Machine\xa0Running\xa0at\xa0P2\n2001\tIndicator\xa0Machine\xa0Error\xa0at\xa0P2\n2002\tIndicator Tower\xa0Lamp\xa0Red\n2003\tIndicator Tower\xa0Lamp\xa0Yellow\n2004\tIndicator Tower\xa0Lamp\xa0Green\n2005\tIndicator Tower\xa0Lamp\xa0Blue\n2006\tIndicator Buzzer\n2007\tIndicator Acknowledge at P2\n2008\tIndicator Auto Mode P2\n2009\tIndicator Manual Mode P2\n2010\t\n2011\t\n2012\t\n2013\t\n2014\t\n2015\tMove Forward for Loaded Pallet Outfeed Roller Conveyor 5 '
  1326 = '2000\tIndicator\xa0Machine\xa0Running\xa0at\xa0P2\n2001\tIndicator\xa0Machine\xa0Error\xa0at\xa0P2\n2002\tIndicator Tower\xa0Lamp\xa0Red\n2003\tIndicator Tower\xa0Lamp\xa0Yellow\n2004\tIndicator Tower\xa0Lamp\xa0Green\n2005\tIndicator Tower\xa0Lamp\xa0Blue\n2006\tIndicator Buzzer\n2007\tIndicator Acknowledge at P2\n2008\tIndicator Auto Mode P2\n2009\tIndicator Manual Mode P2\n2010\t\n2011\t\n2012\t\n2013\t\n2014\t\n2015\tMove Forward for Loaded Pallet Outfeed Roller Conveyor 5 is Running (FC51)'
  1448 = '2000\tIndicator\xa0Machine\xa0Running\xa0at\xa0P2\n2001\tIndicator\xa0Machine\xa0Error\xa0at\xa0P2\n2002\tIndicator Tower\xa0Lamp\xa0Red\n2003\tIndicator Tower\xa0Lamp\xa0Yellow\n2004\tIndicator Tower\xa0Lamp\xa0Green\n2005\tIndicator Tower\xa0Lamp\xa0Blue\n2006\tIndicator Buzzer\n2007\tIndicator Acknowledge at P2\n2008\tIndicator Auto Mode P2\n2009\tIndicator Manual Mode P2\n2010\tStatus Solenoid Door Outfeed\n2011\tStatus Solenoid Door Wrapper\n2012\t\n2013\tPneumatic Stopper Modullar Adv\n2014\tPneumatic Stopper Modullar Rtc\n2015\tMove Forward for Loaded Pallet Outfeed Roller Conveyor 5 '
  313 = '2000 - Indicator\xa0Machine\xa0Running\xa0at\xa0P2'
  1338 = '2001 - Indicator\xa0Machine\xa0Error\xa0at\xa0P2'
  1470 = '2002 - Indicator Tower\xa0Lamp\xa0Red'
  1518 = '2003 - Indicator Tower\xa0Lamp\xa0Yellow'
  354 = '2004 - Indicator Tower\xa0Lamp\xa0Green'
  344 = '2005 - Indicator Tower\xa0Lamp\xa0Blue'
  827 = '2006 - Indicator Buzzer'
  1516 = '2007 - Indicator Acknowledge at P2'
  457 = '2008 - Indicator Auto Mode P2'
  261 = '2009 - Indicator Manual Mode P2'
  1808 = '2010'
  665 = '2011'
  299 = '2012'
  1958 = '2013'
  2028 = '2014'
  296 = '2015 - Move Forward for Loaded Pallet Outfeed Roller Conveyor 5 is Running (FC51)'
  1246 = '20xx'
  1383 = '21'
  999 = '2100\tMove Forward for Transfer Modullar Conveyor  1\n2101\tMove Forward for Transfer Modullar Conveyor  2\n2102\tMove Forward for Transfer Modullar Conveyor  3\n2103\tMove Forward for Transfer Modullar Conveyor  4 \n2104\tMove Forward for Infeed Roller Conveyor\n2105\tMove Forward for Stop & Go Belt Conveyor\n2106\tMove Forward For Buffer Roller  Conveyor 1\n2107\tMove Forward For Buffer Roller  Conveyor 2\n2108\tMove Forward for Loaded Pallet Buffer Conveyor 1 (FC51)\n2109\tMove Forward for Loaded Pallet Outfeed Roller Conveyor 1 (FC51)\n2110\tMove Forward for Right Angel  (FC51)\n2111\tMove Forward for Right Angel Lifter (FC51)\n2112\tMove Forward for Loaded Pallet Outfeed Roller Conveyor (FC51)\n2113\tMove Forward for Loaded Pallet Outfeed Roller Conveyor (FC51)\n2114\tMove Forward for Loaded Pallet Outfeed Roller Conveyor (FC51)\n2115\tReset Error for All Inverter at P2, Relay'
  1554 = '2100 - Move Forward for Transfer Modullar Conveyor  1'
  246 = '2101 - Move Forward for Transfer Modullar Conveyor  2'
  1720 = '2102 - Move Forward for Transfer Modullar Conveyor  3'
  2027 = '2103 - Move Forward for Transfer Modullar Conveyor  4'
  2144 = '2104 - Move Forward for Infeed Roller Conveyor'
  1780 = '2105 - Move Forward for Stop & Go Belt Conveyor'
  789 = '2106 - Move Forward For Buffer Roller  Conveyor 1'
  845 = '2107 - Move Forward For Buffer Roller  Conveyor 2'
  332 = '2108 - Move Forward for Loaded Pallet Buffer Conveyor 1 is Running (FC51)'
  1413 = '2109 - Move Forward for Loaded Pallet Outfeed Roller Conveyor 1 is Running (FC51)'
  2114 = '2110 - Move Forward for Right Angel is Running (FC51)'
  1786 = '2111 - Move Forward for Right Angel Lifter is Running  (FC51)'
  599 = '2112 - Move Forward for Loaded Pallet Outfeed Roller Conveyor 2 is Running (FC51)'
  1417 = '2113 - Move Forward for Loaded Pallet Outfeed Roller Conveyor 3 is Running (FC51)'
  1934 = '2114 - Move Forward for Loaded Pallet Outfeed Roller Conveyor 4 is Running (FC51)'
  1914 = '2115 - Reset Error for All Inverter at P2, Relay'
  5141 = '21xx'
  4073 = '22'
  5246 = '2200\tMove Forward For Loaded Pallet Buffer Conveyor 2 \n2201\t\n2202\tPneumatic Box Stopper 1\n2203\tPneumatic Box Stopper 2\n2204\t\n2205\tPneumatic Pusher Stop & Go  Adv\n2206\tPneumatic Pusher Stop & Go  Rtc\n2207\tPneumatic Pusher Buffer Roller 1 Adv\n2208\tPneumatic Pusher Buffer Roller 1 Rtc\n2209\tPneumatic Pusher Buffer Roller 2 Adv\n2210\tPneumatic Pusher Buffer Roller 2 Rtc\n2211\t\n2212\t\n2213\tRelease Brake Motor Right Angle Lifter\n2214\tInterlock Request Pallet to Infeed Dispenser\n2215\tInterlock Request Pallet to Conveyor Outfeed Existing'
  4704 = '2200\tMove Forward For Loaded Pallet Buffer Conveyor 2 \n2201\t\n2202\tPneumatic Box Stopper 1\n2203\tPneumatic Box Stopper 2\n2204\t\n2205\tPneumatic Pusher Stop & Go  Adv\n2206\tPneumatic Pusher Stop & Go  Rtc\n2207\tPneumatic Pusher Buffer Roller 1 Adv\n2208\tPneumatic Pusher Buffer Roller 1 Rtc\n2209\tPneumatic Pusher Buffer Roller 2 Adv\n2210\tPneumatic Pusher Buffer Roller 2 Rtc\n2211\t\n2212\tInterlock Status Infeed Modullar Busy\n2213\tRelease Brake Motor Right Angle Lifter\n2214\tInterlock Request Pallet to Infeed Dispenser\n2215\tInterlock Request Pallet to Conveyor Outfeed Existing'
  4448 = '2200\tMove Forward for Picking Roller Conveyor\n2201\t\n2202\tMove Forward for Placing At Pallet Roller Conveyor  1\n2203\tMove Forward for Placing At Pallet Roller Conveyor  2\n2204\tMove Forward for Placing At Pallet Roller Conveyor  3\n2205\tMove Forward for Placing At Pallet Roller Conveyor  4\n2206\t\n2207\tMove Reverse for Placing At Pallet Roller Conveyor  1\n2208\tMove Reverse for Placing At Pallet Roller Conveyor  2\n2209\tMove Reverse for Placing At Pallet Roller Conveyor  3\n2210\tMove Reverse for Placing At Pallet Roller Conveyor  4\n2211\t\n2212\t\n2213\t\n2214\t\n2215\tReset Error for All Inverter at P1, Relay'
  1097 = '2200 - Move Forward For Loaded Pallet Buffer Conveyor 2 is running'
  1996 = '2201 - Move Forward For Loaded Pallet Buffer Conveyor 3 is running'
  2234 = '2202 - Pneumatic Box Stopper 1'
  1077 = '2203 - Pneumatic Box Stopper 2'
  1574 = '2204'
  2000 = '2205 - Pneumatic Pusher Stop & Go  Adv'
  2273 = '2206 - Pneumatic Pusher Stop & Go  Rtc'
  1355 = '2207 - Pneumatic Pusher Buffer Roller 1 Adv'
  649 = '2208 - Pneumatic Pusher Buffer Roller 1 Rtc'
  1124 = '2209 - Pneumatic Pusher Buffer Roller 2 Adv'
  1549 = '2210 - Pneumatic Pusher Buffer Roller 2 Rtc'
  1686 = '2211'
  521 = '2212'
  731 = '2213 - Release Brake Motor Right AngleLifter'
  1420 = '2214 - Interlock Request Pallet to Inffed Dispenser Exisiting'
  892 = '2215 - Interlock Request Pallet to Conveyor Outfeed Existing'
  2522 = '2222'
  3251 = '22xx'
  1871 = '23'
  2730 = '2300\tIndicator\xa0Machine\xa0Running\xa0at\xa0Dispenser\n2301\tIndicator\xa0Machine\xa0Error\xa0at\xa0Dispenser\n2302\tIndicator\xa0Acknowledge\xa0at\xa0Dispenser\n2303\tIndicator Auto at Dispenser\n2304\tIndicator Manual at Dispenser\n2305\tPallet In Before Wrapper Ready\n2306\tAfter Wrapper Ready to Receive\n2307\tEnd of Transfer Pallet in Outfeed\n2308\tBypass Wrapping\n2309\tRelease Solenoid Door 1 (Outfeed)\n2310\tRelease Solenoid Door 2 (Wrapper)\n2311\tMove Forward for Automatic Pallet Dispenser\n2312\tPneumatic Vertical Up\n2313\tPneumatic Vertical Down\n2314\tPneumatic Horizontal Rectract\n2315\tPneumatic Horizontal Advanced'
  2886 = '2300\tPneumatic Box Centering\n2301\tPneumatic Gap Maker Box Adv\n2302\tPneumatic Gap Maker Box Rtc\n2303\t\n2304\t\n2305\t\n2306\t\n2307\t\n2308\t\n2309\tPneumatic Stopper Transfer\n2310\t\n2311\t\n2312\t\n2313\t\n2314\tStatus Solenoid Door Robot\n2315\tRelease Solenoid Door Robot'
  1960 = '23xx'
  2858 = '24'
  2657 = '2420'
  716 = '2424'
  2290 = '24xx'
  267 = '3'
  234 = '4'
  2507 = '5'
  1978 = '5000\tFeedback Empty pallet shuttle is Running\n5001\tFeedback Load pallet shuttle is Running\n5002\tFeedback Drive Shuttle is Running\n5003\tFeedback Relay Enable STO Conveyor Channel 1\n5004\tPSR To Detect Front Pallet at Empty Pallet Shuttle\n5005\tPSR To Detect Back Pallet at Empty Pallet Shuttle\n5006\tPSR To Detect End Of Front Pallet at Empty Pallet Shuttle\n5007\t\n5008\tPSR To Detect Front Pallet at Load Pallet Shuttle \n5009\tPSR To Detect Back Pallet at Load Pallet Shuttle\n5010\tPSR To Detect End Of Front Pallet at Load Pallet Shuttle \n5011\tPSR To Detect End Of Back Pallet at Load Pallet Shuttle\n5012\tLimit Switch To Detect Left Limit Area\n5013\tLimit Switch To Detect Right Limit Area\n5014\tPRX to Detect Left Limit Area\n5015\tPRX to Detect Right Limit Area'
  2755 = '5000\tFeedback Empty pallet shuttle is Running (FC51-0.75kW)\n5001\tFeedback Load pallet shuttle is Running (FC51-1.5kW)\n5002\tFeedback Drive Shuttle is Running (FC302-2kW)\n5003\tFeedback Relay Enable STO Conveyor Channel 1\n5004\tPSR To Detect Front Pallet at Empty Pallet Shuttle (GL6-P4212)\n5005\tPSR To Detect Back Pallet at Empty Pallet Shuttle (GL6-P4212)\n5006\tPSR To Detect End Of Front Pallet at Empty Pallet Shuttle (GTE6-P4212)\n5007\t\n5008\tPSR To Detect Front Pallet at Load Pallet Shuttle (GL6-P4212)\n5009\tPSR To Detect Back Pallet at Load Pallet Shuttle (GL6-P4212)\n5010\tPSR To Detect End Of Front Pallet at Load Pallet Shuttle (GTE6-P4212)\n5011\tPSR To Detect End Of Back Pallet at Load Pallet Shuttle (GTE6-P4212)\n5012\tLimit Switch To Detect Left Limit Area\n5013\tLimit Switch To Detect Right Limit Area\n5014\tPRX to Detect Left Limit Area (E2B-M30LN30-M1-B2)\n5015\tPRX to Detect Right Limit Area (E2B-M30LN30-M1-B2)'
  4279 = '50xx'
  1699 = '6'
  2740 = '6000\tMove Forward for Empty pallet shuttle\n6001\tMove Forward for Load pallet shuttle\n6002\tMove Reverse for Load pallet shuttle\n6003\tMove Forward for Drive Shuttle\n6004\tMove Reverse for Drive Shuttle\n6005\t\n6006\t\n6007\tReset Error for All Inverter at P2, Relay\n6008\tRelay for Brake Forward\n6009\tRelay for Brake Reverse\n6010\t\n6011\t\n6012\t\n6013\t\n6014\t\n6015\t'
  4443 = '60xx'
  2772 = '7'
  793 = '8'
  1963 = '9'
  443 = 'Acknowladge'
  1278 = 'Active'
  3551 = 'Actual Pos'
  218 = 'Admin'
  4559 = 'ALARM'
  1025 = 'Alarm'
  1909 = 'alarm'
  1685 = 'Alarm Active'
  822 = 'Alarm History'
  102 = 'B1'
  1624 = 'B2'
  2041 = 'Barcode'
  1696 = 'barcode'
  2156 = 'Barcode 1 : %i'
  1844 = 'Barcode 1: %i'
  5201 = 'Barcode 2 : %i'
  3147 = 'Barcode 3 : %i'
  1793 = 'Barcode 4 : %i'
  2969 = 'Barcode Bac : %i'
  3336 = 'Barcode Back Right : %i'
  4029 = 'Barcode Front : %i'
  117 = 'Barcode Front Right : %i'
  2091 = 'Barcode Line '
  698 = 'Barcode Line 1'
  2261 = 'Barcode Line 2'
  2453 = 'Barcode Line 3'
  2195 = 'Barcode Line 4'
  1592 = 'Barcode Product'
  4820 = 'Barcode Result'
  5815 = 'Barcode State'
  2506 = 'Big'
  1054 = 'Buffer 1'
  1788 = 'Buffer 2'
  1550 = 'Bypass'
  916 = 'Bypass FGHS'
  1060 = 'Bypass Wrapper'
  98 = 'Bypass Wrapper Existing'
  740 = 'Cancel'
  4223 = 'Centering'
  1810 = 'Centering Adv'
  2399 = 'Check Buffer 1'
  347 = 'Check Buffer 2'
  1949 = 'Check Dispenser'
  2219 = 'Check Empty'
  2594 = 'Check Infeed'
  1293 = 'Check Load'
  1015 = 'Check Outfee 4'
  3111 = 'Check Outfeed 1'
  1919 = 'Check Outfeed 2'
  802 = 'Check Outfeed 3'
  4075 = 'Check Outfeed 4'
  1895 = 'Check Outfeed 5'
  3153 = 'Check Outfese 4'
  2887 = 'Check Picking'
  3465 = 'Check Placing 1'
  509 = 'Check Placing 2'
  3539 = 'Check Placing 3'
  2157 = 'Check Placing 4'
  3596 = 'Check Stop & Go'
  3957 = 'Check Stopper 1'
  120 = 'Check Stopper 2'
  1645 = 'Code Variant'
  996 = 'Completed'
  787 = 'Control'
  293 = 'Conveyor Off'
  29 = 'Conveyor On'
  1073 = 'Counter'
  1017 = 'COUNTER LINE'
  1285 = 'Counter Placing'
  1257 = 'Current'
  4868 = 'Current Job :'
  2140 = 'CURRENT OFFSET'
  2714 = 'CURRENT USAGE OFFSET'
  2098 = 'CURRENT USAGE PRODUCT'
  1369 = 'CURRENT USAGE PRODUCT LINE A :'
  908 = 'Data Pallet'
  2246 = 'Data Pallet 1'
  1929 = 'Data Pallet 2'
  1279 = 'Data Pallet 3'
  1737 = 'Data Pallet 4'
  4164 = 'Data Production'
  1564 = 'Data_GVL.dt_OEETime.Precentage[0].Running'
  3001 = 'Date & Time : %s'
  1567 = 'Delay'
  297 = 'Delay\nModullar Off'
  1559 = 'Delay \nModullar On'
  363 = 'Delay Brake'
  1968 = 'Delay Centering'
  4478 = 'Delay Modullar On'
  25 = 'Delay RA Lifter'
  1796 = 'Delay RA Release'
  5620 = 'DI\n2'
  3664 = 'DI\n3'
  6930 = 'DI \n1'
  1399 = 'DI \n4'
  1228 = 'DI \n5'
  3034 = 'Disable Overflow'
  600 = 'Dispenser'
  1051 = 'Dispenser %s'
  3292 = 'Dispenser Pos'
  8057 = 'DO\n1'
  6203 = 'DO\n2'
  5936 = 'DO \n3'
  132 = 'Download'
  1053 = 'Drive Fwd'
  616 = 'Drive Rev'
  1184 = 'EAN'
  640 = 'EAN Variant'
  1701 = 'Edit'
  153 = 'EDIT OFFSET'
  1541 = 'Empty Fwd'
  1959 = 'Enable Overflow'
  1398 = 'Error'
  30 = 'Error Message'
  1845 = 'FGHS'
  336 = 'Flsuhed'
  3608 = 'Flushed'
  1957 = 'Flushing'
  2119 = 'Gap Maker Adv'
  3605 = 'Gap Maker Rtc'
  1301 = 'H - 1'
  729 = 'H - 2'
  1725 = 'H - 3'
  3378 = 'H - 4'
  1131 = 'H - 5'
  984 = 'H - 6'
  1620 = 'Height'
  1179 = 'History'
  294 = 'Home'
  4586 = 'Horizontal Adv'
  212 = 'Horizontal Rtc'
  927 = 'I/O'
  3976 = 'I/O Status'
  2384 = 'Infeed'
  693 = 'Infeed %s'
  4819 = 'Input 1'
  788 = 'Input/Ouput'
  3950 = 'Jog Speed'
  1724 = 'Layer'
  810 = 'Length'
  938 = 'Line'
  345 = 'Line 1'
  1646 = 'Line 2'
  2103 = 'Line 3'
  949 = 'Line 4'
  754 = 'Line1'
  1086 = 'Link Up'
  2922 = 'Load'
  1652 = 'Load Fwd'
  376 = 'Load Rev'
  1249 = 'Lock Modullar'
  3929 = 'Login'
  636 = 'Logout'
  3068 = 'Machine'
  823 = 'MACHINE ERROR'
  311 = 'Machine Error '
  2545 = 'Machine Performance'
  214 = 'Machine Status'
  237 = 'Machine Status : '
  264 = 'Manual / Auto'
  191 = 'Manual Mode'
  2036 = 'Max Speed'
  4387 = 'Message'
  3703 = 'Message :'
  3801 = 'Min Speed'
  655 = 'Modullar Off'
  3500 = 'Modullar On'
  1916 = 'Motor'
  2414 = 'Motor Buffer 1'
  3580 = 'Motor Buffer 2'
  1687 = 'Motor Dispenser'
  3476 = 'Motor Drive'
  1995 = 'Motor Empty'
  1999 = 'Motor Infeed'
  1009 = 'Motor Load'
  1570 = 'Motor Modullar 1'
  2461 = 'Motor Modullar 2'
  3914 = 'Motor Modullar 3'
  2266 = 'Motor Modullar 4'
  1584 = 'Motor Outfeed 1'
  1578 = 'Motor Outfeed 2'
  4128 = 'Motor Outfeed 3'
  2996 = 'Motor Outfeed 4'
  2213 = 'Motor Outfeed 5'
  806 = 'Motor Picking'
  1308 = 'Motor Placing'
  4083 = 'Motor Placing 1'
  3756 = 'Motor Placing 2'
  1538 = 'Motor Placing 3'
  3434 = 'Motor Placing 4'
  2865 = 'Motor Stop & Go'
  3798 = 'MTBF'
  928 = 'MTBF Dispenser'
  1673 = 'MTBF Infeed'
  3582 = 'MTBF Outfeed'
  2620 = 'MTBF Picking'
  4025 = 'MTBF Placing'
  3737 = 'MTBF Shuttle'
  971 = 'Mute Buzzer'
  1698 = 'Name'
  2988 = 'None'
  1931 = 'O1'
  1900 = 'O2'
  2151 = 'O3'
  248 = 'O4'
  427 = 'O5'
  2089 = 'OEE'
  544 = 'oFFSET'
  1531 = 'Offset'
  1241 = 'Offset Pos'
  1192 = 'Operator'
  765 = 'Outfeed'
  1586 = 'Outfeed %s'
  1157 = 'Outfeed 1'
  2278 = 'Outfeed 2'
  353 = 'Outfeed 3'
  1683 = 'Outfeed 4'
  1234 = 'Outfeed 5'
  3206 = 'Outfeed Pos'
  38 = 'Outfeed System'
  1547 = 'Pallet'
  753 = 'Pallet 1'
  828 = 'Pallet 2'
  346 = 'Pallet 3'
  703 = 'Pallet 4'
  512 = 'Pallet ID'
  105 = 'Panel 2\n(Outfeed)'
  3221 = 'Panel Outfeed'
  1688 = 'Panel Robot'
  630 = 'Panel Shuttle'
  1177 = 'PARAMETER'
  774 = 'Parameter'
  2249 = 'Parameter Dispenser'
  2946 = 'Parameter Infeed'
  868 = 'Parameter Outfeed'
  3443 = 'Parameter Picking'
  4220 = 'Parameter Placing'
  1857 = 'Parameter Shuttle'
  2258 = 'Paramter Dispenser'
  2362 = 'Paramter Infeed'
  847 = 'Paramter Shuttle'
  2032 = 'Pattern'
  1794 = 'Performance'
  5370 = 'Pick'
  623 = 'Picking'
  1976 = 'Picking %s'
  2848 = 'Pickint'
  2685 = 'Place 1'
  871 = 'Place 1 %s'
  3699 = 'Place 1 Empty'
  2324 = 'Place 1 Fwd'
  915 = 'Place 1 Load'
  2419 = 'Place 1 Rev'
  3052 = 'Place 2'
  1296 = 'Place 2 %s'
  513 = 'Place 2 Empty'
  594 = 'Place 2 Fwd'
  2179 = 'Place 2 Load'
  798 = 'Place 2 Rev'
  1170 = 'Place 3'
  1456 = 'Place 3 %s'
  1859 = 'Place 3 Empty'
  1838 = 'Place 3 Fwd'
  805 = 'Place 3 Load'
  1336 = 'Place 3 Rev'
  921 = 'Place 4'
  1523 = 'Place 4 %s'
  284 = 'Place 4 Empty'
  846 = 'Place 4 Fwd'
  2001 = 'Place 4 Load'
  1466 = 'Place 4 Rev'
  3435 = 'Place1 Load'
  2921 = 'Place21 Load'
  2975 = 'Placing'
  2287 = 'Placing %s'
  1374 = 'Placing 1'
  2353 = 'Placing 1 %s'
  2357 = 'Placing 2'
  2319 = 'Placing 2 %s'
  1987 = 'Placing 3'
  2262 = 'Placing 3 %s'
  1439 = 'Placing 4'
  1795 = 'Placing 4 %s'
  1588 = 'Planned'
  531 = 'PLC Status'
  717 = 'PLC STATUS '
  3853 = 'Pneumatic'
  941 = 'Product'
  41 = 'Product Info List'
  1506 = 'PRODUCT INFO LIST'
  5401 = 'Production'
  2337 = 'Pusher \nBuffer 1 Adv'
  1856 = 'Pusher \nBuffer 1 Rtc'
  3650 = 'Pusher \nBuffer 2 Adv'
  3533 = 'Pusher \nBuffer 2 Rtc'
  2872 = 'Pusher Buffer 1 Adv'
  3220 = 'Pusher Buffer 1 Rtc'
  3079 = 'Pusher Buffer 2 Adv'
  3786 = 'Pusher Buffer 2 Rtc'
  482 = 'Pusher Infeed'
  1983 = 'Pusher Stop \n& Go Adv'
  1126 = 'Pusher Stop \n& Go Rtc'
  4673 = 'Pusher Stop & Go'
  3186 = 'Pusher Stop & Go Adv'
  2573 = 'Pusher Stop & Go Rtc'
  824 = 'RA Delay'
  911 = 'RA Lifter'
  953 = 'RA Transfer'
  2104 = 'Recipe'
  1395 = 'Recipe Line 1'
  605 = 'Recipe Line 2'
  1275 = 'Recipe Line 3'
  794 = 'Recipe Line 4'
  3778 = 'Reject'
  2040 = 'REJECT FULL'
  5185 = 'Reject History'
  3156 = 'Reject ID'
  543 = 'Release Brake Right Angle'
  2281 = 'Reset'
  597 = 'Reset Link Up'
  2475 = 'Right Angle'
  1702 = 'Robot'
  593 = 'Robot %s'
  1008 = 'Robotic'
  15 = 'Rotate'
  485 = 'Run'
  441 = 'Running'
  1614 = 'Save'
  45 = 'Seq Index   :'
  766 = 'Sequence Machine'
  2004 = 'Service'
  825 = 'Shift - 1'
  2122 = 'Shift - 2'
  492 = 'Shift - 3'
  1492 = 'Shift1'
  259 = 'Shuttl e%s'
  1982 = 'Shuttle'
  256 = 'Shuttle %s'
  1055 = 'Shuttle Fwd'
  1240 = 'Shuttle Pos : '
  458 = 'Shuttle Pos : %i'
  1911 = 'Shuttle Postion'
  628 = 'Shuttle Rev'
  2253 = 'Shuttle Speed'
  4529 = 'Small'
  217 = 'Standby'
  538 = 'State Machine'
  2943 = 'Statistic'
  1757 = 'Statistic Outfeed'
  4484 = 'Statistic Production'
  2443 = 'Statistic Robot'
  172 = 'Statistic RObot'
  1760 = 'Status'
  542 = 'STATUS'
  340 = 'Stop'
  2359 = 'Stop & Go'
  2447 = 'Stopped'
  395 = 'Stopper 1'
  3325 = 'Stopper 1 Adv'
  3749 = 'Stopper 2'
  370 = 'Stopper 2 Adv'
  464 = 'Test Infeed'
  1147 = 'TEST MODE'
  2350 = 'Test Outfeed'
  3298 = 'Test Picking'
  2118 = 'Test Place 1'
  1889 = 'Test Place 2'
  2025 = 'Test Place 3'
  143 = 'Test Place 4'
  1360 = 'Test Shuttle'
  187 = 'Time'
  31 = 'Time Stop'
  32 = 'Timer'
  1619 = 'Today'
  379 = 'Upload'
  3233 = 'Username : %s'
  103 = 'Variant'
  317 = 'Vertical Rtc'
  4347 = 'Vertval Adv'
  1444 = 'Width'
  4697 = 'Wiring No. :'
  1276 = 'X'
  801 = 'Y'
END_TEXTLIST

// ---- VISUs/FGHS/DataPallet2.TcVIS
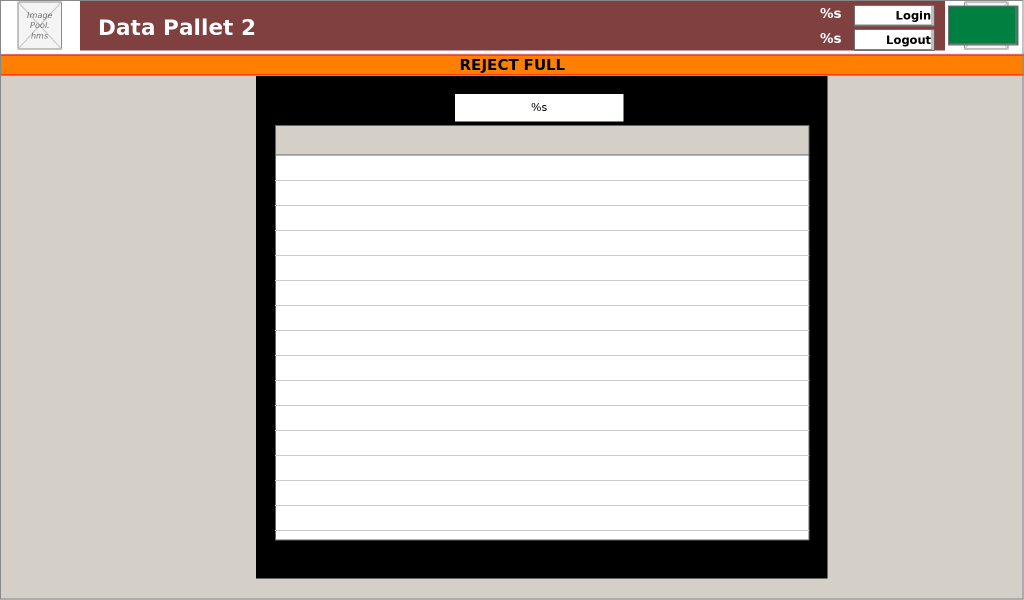
VISUALIZATION DataPallet2  // 1024x600
    Frame (0,-2 1021x55)
        shows Header()
    Label (95,15 250x25), "Data Pallet 2"
    RoundedRectangle (256,76 571x502)
    Table (275,125 534x415), data array: Status_GVL.arDataPallet2
        p3854506369: Status_GVL.arDataPallet2[INDEX].BarcodePallet
        p1892666644: Status_GVL.arDataPallet2[INDEX].BarcodePalletTime
        p338671338: Status_GVL.arPalletizingBuffer[1].EANVariant
        p2170511999: Status_GVL.arPalletizingBuffer[1].CodeVariant
        p3723444502: Status_GVL.arPalletizingBuffer[1].ProductDescription
        p1218418051: Status_GVL.arPalletizingBuffer[1].PalletCreationDate
        p746581629: Status_GVL.arPalletizingBuffer[1].BarcodeProduct
        p3104783080: Status_GVL.arPalletizingBuffer[1].BarcodeProductTime
    RoundedRectangle (454,93 170x29), "%s", text variable: Status_GVL.arPalletID[2]
END_VISUALIZATION

// ---- VISUs/FGHS/DataPallet3.TcVIS
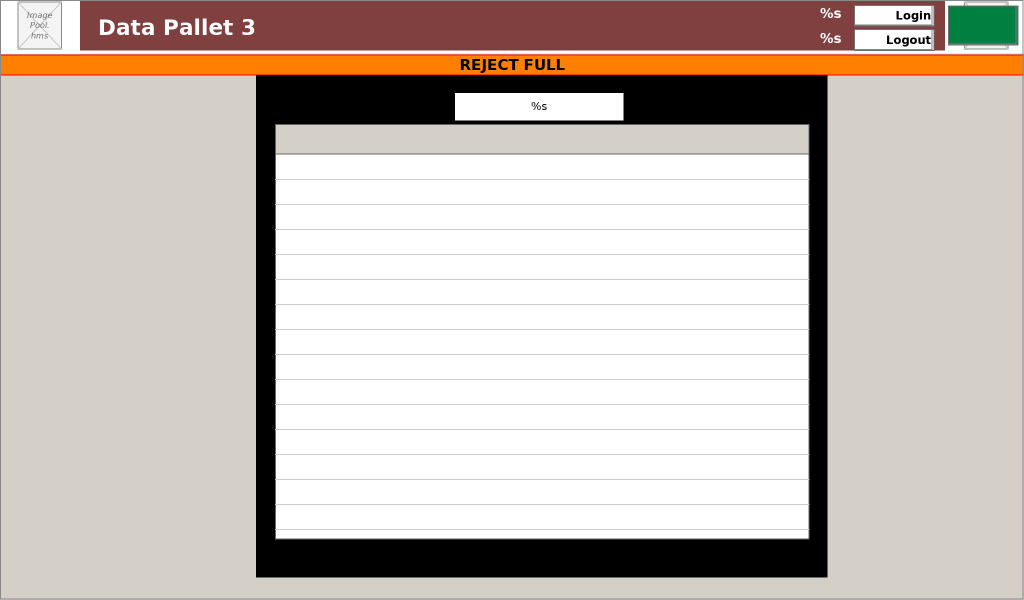
VISUALIZATION DataPallet3  // 1024x600
    Frame (0,-2 1021x55)
        shows Header()
    Label (95,15 250x25), "Data Pallet 3"
    RoundedRectangle (256,75 571x502)
    Table (275,124 534x415), data array: Status_GVL.arDataPallet3
        p3854506369: Status_GVL.arDataPallet3[INDEX].BarcodePallet
        p1892666644: Status_GVL.arDataPallet3[INDEX].BarcodePalletTime
        p338671338: Status_GVL.arPalletizingBuffer[1].EANVariant
        p2170511999: Status_GVL.arPalletizingBuffer[1].CodeVariant
        p3723444502: Status_GVL.arPalletizingBuffer[1].ProductDescription
        p1218418051: Status_GVL.arPalletizingBuffer[1].PalletCreationDate
        p746581629: Status_GVL.arPalletizingBuffer[1].BarcodeProduct
        p3104783080: Status_GVL.arPalletizingBuffer[1].BarcodeProductTime
    RoundedRectangle (454,92 170x29), "%s", text variable: Status_GVL.arPalletID[3]
END_VISUALIZATION

// ---- VISUs/FGHS/DataPallet4.TcVIS
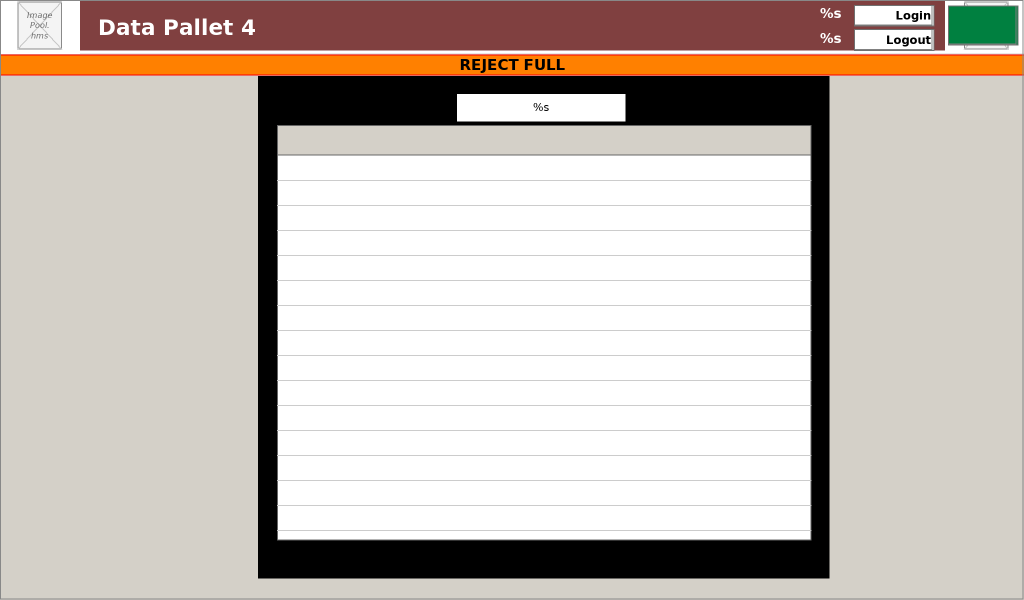
VISUALIZATION DataPallet4  // 1024x600
    Frame (0,-2 1021x55)
        shows Header()
    Label (95,15 250x25), "Data Pallet 4"
    RoundedRectangle (258,76 571x502)
    Table (277,125 534x415), data array: Status_GVL.arDataPallet4
        p3854506369: Status_GVL.arDataPallet4[INDEX].BarcodePallet
        p1892666644: Status_GVL.arDataPallet4[INDEX].BarcodePalletTime
        p338671338: Status_GVL.arPalletizingBuffer[1].EANVariant
        p2170511999: Status_GVL.arPalletizingBuffer[1].CodeVariant
        p3723444502: Status_GVL.arPalletizingBuffer[1].ProductDescription
        p1218418051: Status_GVL.arPalletizingBuffer[1].PalletCreationDate
        p746581629: Status_GVL.arPalletizingBuffer[1].BarcodeProduct
        p3104783080: Status_GVL.arPalletizingBuffer[1].BarcodeProductTime
    RoundedRectangle (456,93 170x29), "%s", text variable: Status_GVL.arPalletID[4]
END_VISUALIZATION

// ---- VISUs/FGHS/FGHS.TcVIS
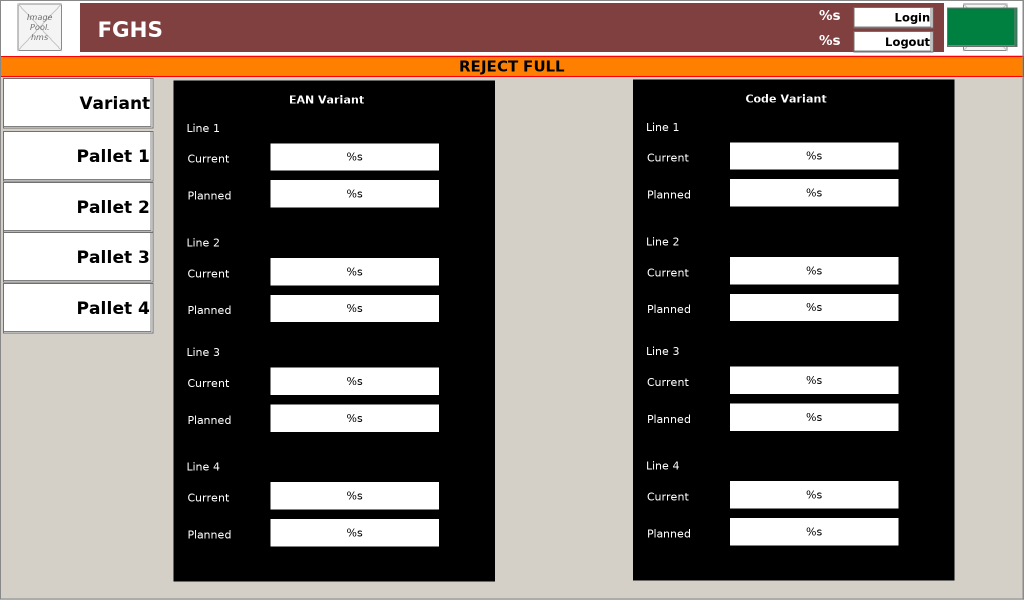
VISUALIZATION FGHS  // 1024x600
    Frame (0,2 1023x598)
        shows FGHS_1()
        shows DataPallet1()
        shows DataPallet2()
        shows DataPallet3()
        shows DataPallet4()
    Button (3,78 150x50), "Variant", image: VisuSymbols.Symbols.Database2
        OnMouseDown: FrameSelectionChange Selection=SelectedFrame=146e207b-fd78-4676-ba16-384fa245d7d2, GlobSel=AssignDir=MainPage.GenElemInst_1003, AssignType=Directly, SelType=Locally
    Button (3,131 150x50), "Pallet 1", image: VisuSymbols.Symbols.Database2
        OnMouseDown: FrameSelectionChange Selection=SelectedFrame=146e207b-fd78-4676-ba16-384fa245d7d2, Selection=1, GlobSel=AssignDir=MainPage.GenElemInst_1003, AssignType=Directly, SelType=Locally
    Button (3,182 150x50), "Pallet 2", image: VisuSymbols.Symbols.Database2
        OnMouseDown: FrameSelectionChange Selection=SelectedFrame=146e207b-fd78-4676-ba16-384fa245d7d2, Selection=2, GlobSel=AssignDir=MainPage.GenElemInst_1003, AssignType=Directly, SelType=Locally
    Button (3,232 150x50), "Pallet 3", image: VisuSymbols.Symbols.Database2
        OnMouseDown: FrameSelectionChange Selection=SelectedFrame=146e207b-fd78-4676-ba16-384fa245d7d2, Selection=3, GlobSel=AssignDir=MainPage.GenElemInst_1003, AssignType=Directly, SelType=Locally
    Button (3,283 150x50), "Pallet 4", image: VisuSymbols.Symbols.Database2
        OnMouseDown: FrameSelectionChange Selection=SelectedFrame=146e207b-fd78-4676-ba16-384fa245d7d2, Selection=4, GlobSel=AssignDir=MainPage.GenElemInst_1003, AssignType=Directly, SelType=Locally
END_VISUALIZATION

// ---- VISUs/FGHS/FGHS_1.TcVIS
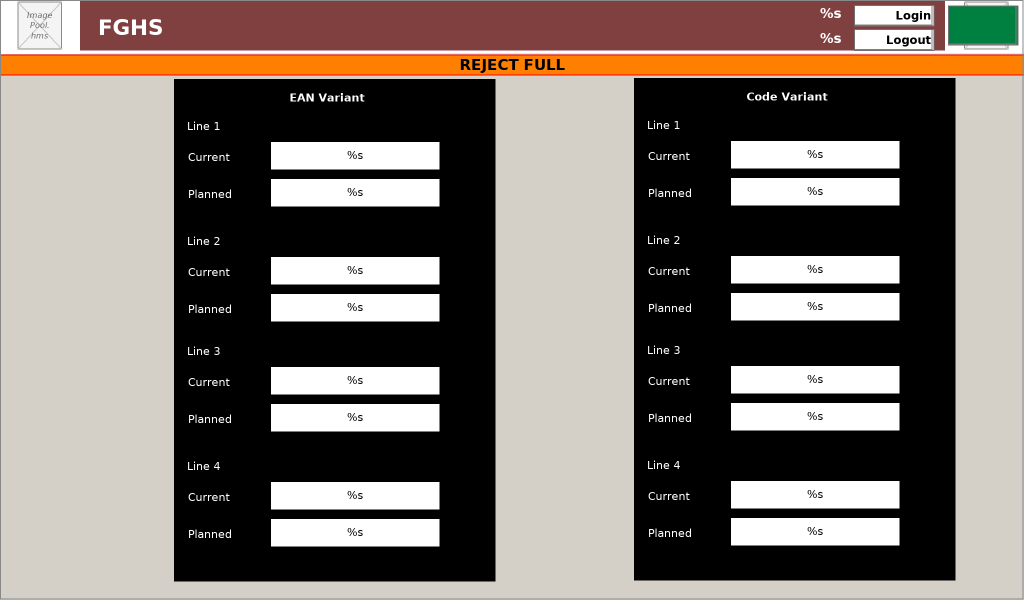
VISUALIZATION FGHS_1  // 1024x600
    Frame (0,-2 1021x55)
        shows Header()
    RoundedRectangle (174,79 321x502)
    Label (214,78 227x40), "EAN Variant"
    Label (185,140 78x35), "Current"
    RoundedRectangle (270,141 170x29), "%s", text variable: Status_GVL.arCurrent_EAN[1]
        OnMouseClick: write Status_GVL.RecipeLine[1].EANVariant via Default
    Label (185,177 78x35), "Planned"
    RoundedRectangle (270,178 170x29), "%s", text variable: Status_GVL.arPlanned_EAN[1]
    Label (95,15 250x25), "FGHS"
    Label (184,109 78x35), "Line 1"
    Label (185,255 78x35), "Current"
    RoundedRectangle (270,256 170x29), "%s", text variable: Status_GVL.arCurrent_EAN[2]
        OnMouseClick: write Status_GVL.RecipeLine[2].EANVariant via Default
    Label (185,292 78x35), "Planned"
    RoundedRectangle (270,293 170x29), "%s", text variable: Status_GVL.arPlanned_EAN[2]
    Label (184,224 78x35), "Line 2"
    Label (185,365 78x35), "Current"
    RoundedRectangle (270,366 170x29), "%s", text variable: Status_GVL.arCurrent_EAN[3]
        OnMouseClick: write Status_GVL.RecipeLine[3].EANVariant via Default
    Label (185,402 78x35), "Planned"
    RoundedRectangle (270,403 170x29), "%s", text variable: Status_GVL.arPlanned_EAN[3]
    Label (184,334 78x35), "Line 3"
    Label (185,480 78x35), "Current"
    RoundedRectangle (270,481 170x29), "%s", text variable: Status_GVL.arCurrent_EAN[4]
        OnMouseClick: write Status_GVL.RecipeLine[4].EANVariant via Default
    Label (185,517 78x35), "Planned"
    RoundedRectangle (270,518 170x29), "%s", text variable: Status_GVL.arPlanned_EAN[4]
    Label (184,449 78x35), "Line 4"
    RoundedRectangle (634,78 321x502)
    Label (674,77 227x40), "Code Variant"
    Label (645,139 78x35), "Current"
    RoundedRectangle (730,140 170x29), "%s", text variable: Status_GVL.arCurrent_CodeVariant[1]
        OnMouseClick: write Status_GVL.RecipeLine[1].CodeVariant via Default
    Label (645,176 78x35), "Planned"
    RoundedRectangle (730,177 170x29), "%s", text variable: Status_GVL.arPlanned_CodeVariant[1]
    Label (644,108 78x35), "Line 1"
    Label (645,254 78x35), "Current"
    RoundedRectangle (730,255 170x29), "%s", text variable: Status_GVL.arCurrent_CodeVariant[2]
        OnMouseClick: write Status_GVL.RecipeLine[2].CodeVariant via Default
    Label (645,291 78x35), "Planned"
    RoundedRectangle (730,292 170x29), "%s", text variable: Status_GVL.arPlanned_CodeVariant[2]
    Label (644,223 78x35), "Line 2"
    Label (645,364 78x35), "Current"
    RoundedRectangle (730,365 170x29), "%s", text variable: Status_GVL.arCurrent_CodeVariant[3]
        OnMouseClick: write Status_GVL.RecipeLine[3].CodeVariant via Default
    Label (645,401 78x35), "Planned"
    RoundedRectangle (730,402 170x29), "%s", text variable: Status_GVL.arPlanned_CodeVariant[3]
    Label (644,333 78x35), "Line 3"
    Label (645,479 78x35), "Current"
    RoundedRectangle (730,480 170x29), "%s", text variable: Status_GVL.arCurrent_CodeVariant[4]
        OnMouseClick: write Status_GVL.RecipeLine[4].CodeVariant via Default
    Label (645,516 78x35), "Planned"
    RoundedRectangle (730,517 170x29), "%s", text variable: Status_GVL.arPlanned_CodeVariant[4]
    Label (644,448 78x35), "Line 4"
END_VISUALIZATION

// ---- VISUs/FGHS/DataPallet1.TcVIS
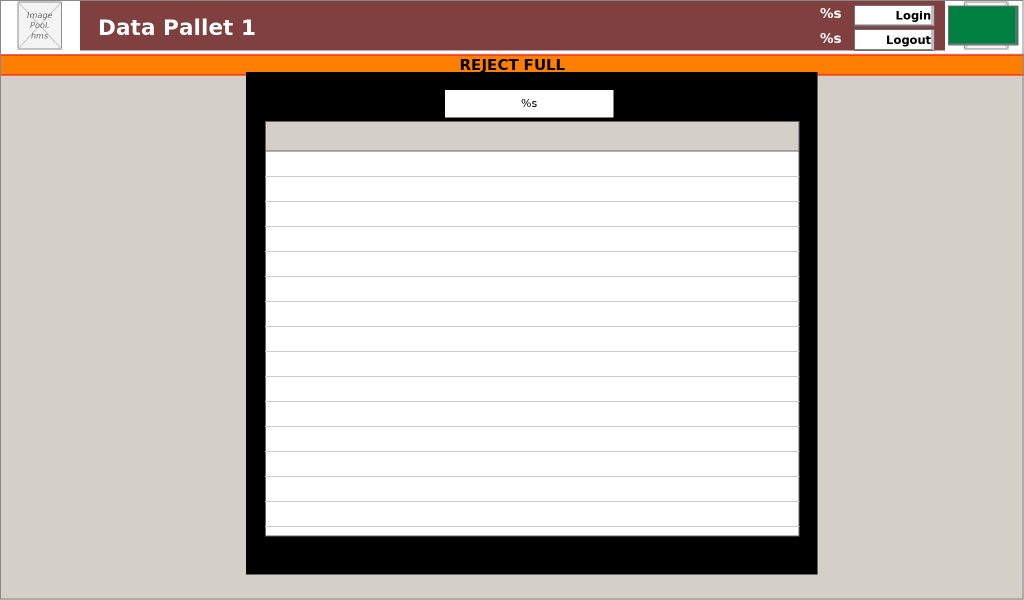
VISUALIZATION DataPallet1  // 1024x600
    Frame (0,-2 1021x55)
        shows Header()
    RoundedRectangle (246,72 571x502)
    Label (95,15 250x25), "Data Pallet 1"
    Table (265,121 534x415), data array: Status_GVL.arDataPallet1
        p3854506369: Status_GVL.arDataPallet1[INDEX].BarcodePallet
        p1892666644: Status_GVL.arDataPallet1[INDEX].BarcodePalletTime
        p338671338: Status_GVL.arPalletizingBuffer[1].EANVariant
        p2170511999: Status_GVL.arPalletizingBuffer[1].CodeVariant
        p3723444502: Status_GVL.arPalletizingBuffer[1].ProductDescription
        p1218418051: Status_GVL.arPalletizingBuffer[1].PalletCreationDate
        p746581629: Status_GVL.arPalletizingBuffer[1].BarcodeProduct
        p3104783080: Status_GVL.arPalletizingBuffer[1].BarcodeProductTime
    RoundedRectangle (444,89 170x29), "%s", text variable: Status_GVL.arPalletID[1]
END_VISUALIZATION

// ---- VISUs/Main/Alarm/RejectMsg.TcVIS
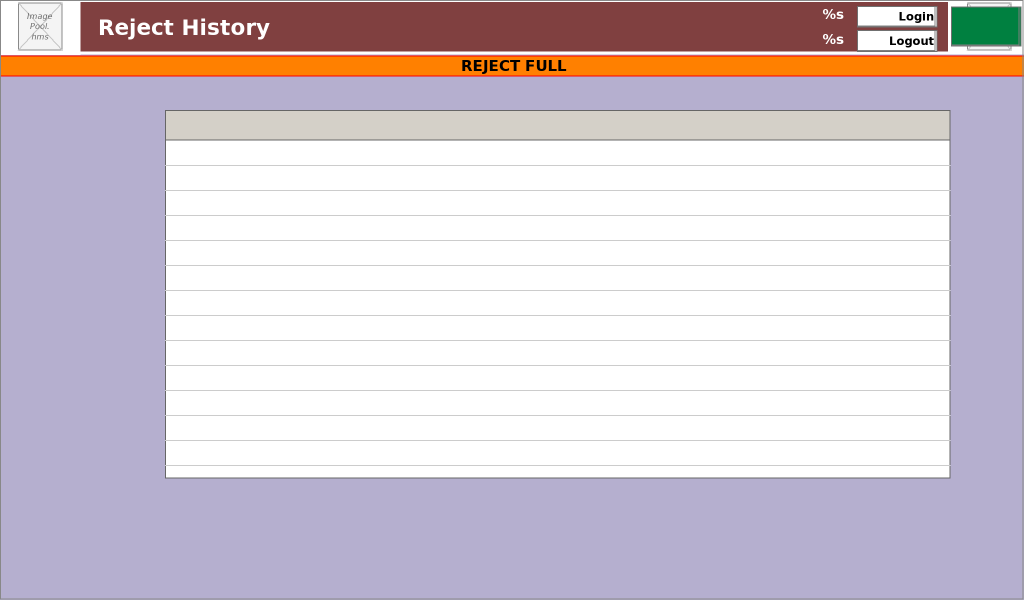
VISUALIZATION RejectMsg  // 1024x600
    Frame (0,-1 1024x55)
        shows Header()
    Label (95,15 250x25), "Reject History"
    Table (165,110 785x368), data array: Status_GVL.arRejectMsg
        p3854506369: Status_GVL.arRejectMsg[INDEX].Status
        p1892666644: Status_GVL.arRejectMsg[INDEX].RejectID
        p338671338: Status_GVL.arRejectMsg[INDEX].RejectType
        p2170511999: Status_GVL.arRejectMsg[INDEX].Counter
        p511219082: Reject ID
        p3723444502: Status_GVL.arRejectMsg[INDEX].RejectMsg
        p1218418051: Status_GVL.arRejectMsg[INDEX].Timestamp
        p2237128397: Message
END_VISUALIZATION

// ---- VISUs/Main/Alarm/AlarmHistory.TcVIS
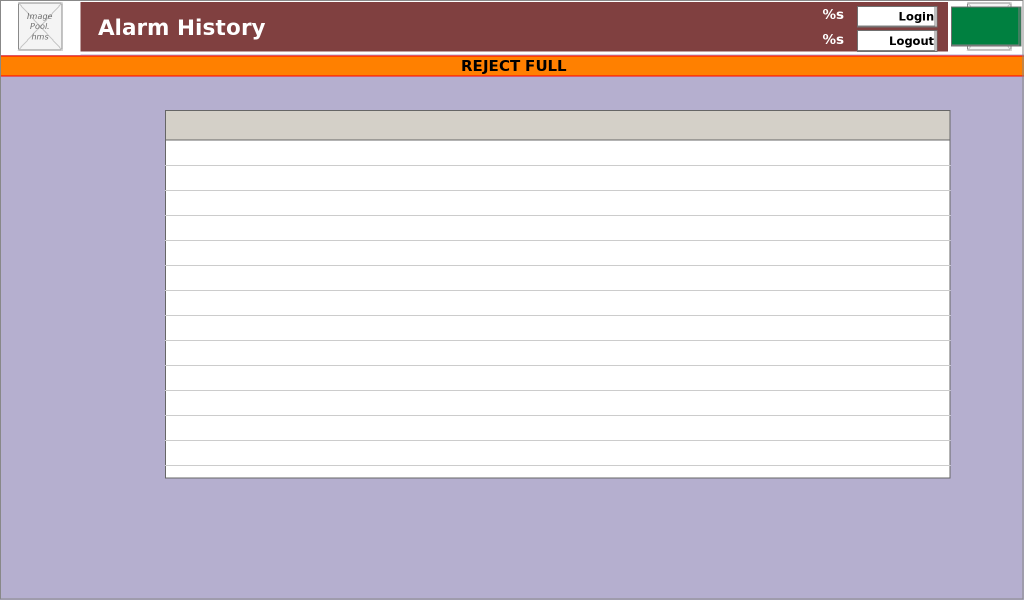
VISUALIZATION AlarmHistory  // 1024x600
    Frame (0,-1 1024x55)
        shows Header()
    Label (95,15 250x25), "Alarm History"
    Table (165,110 785x368), data array: status_Gvl.arAlarmHistory
        p3854506369: status_Gvl.arAlarmHistory[INDEX].Status
        p1892666644: status_Gvl.arAlarmHistory[INDEX].ErrorID
        p338671338: status_Gvl.arAlarmHistory[INDEX].ErrorMsg
        p2170511999: status_Gvl.arAlarmHistory[INDEX].TimeStop
        p511219082: Error ID
        p1755163831: Error Message
        p4092479075: Time Stop
END_VISUALIZATION

// ---- VISUs/Main/Alarm/AlarmActive.TcVIS
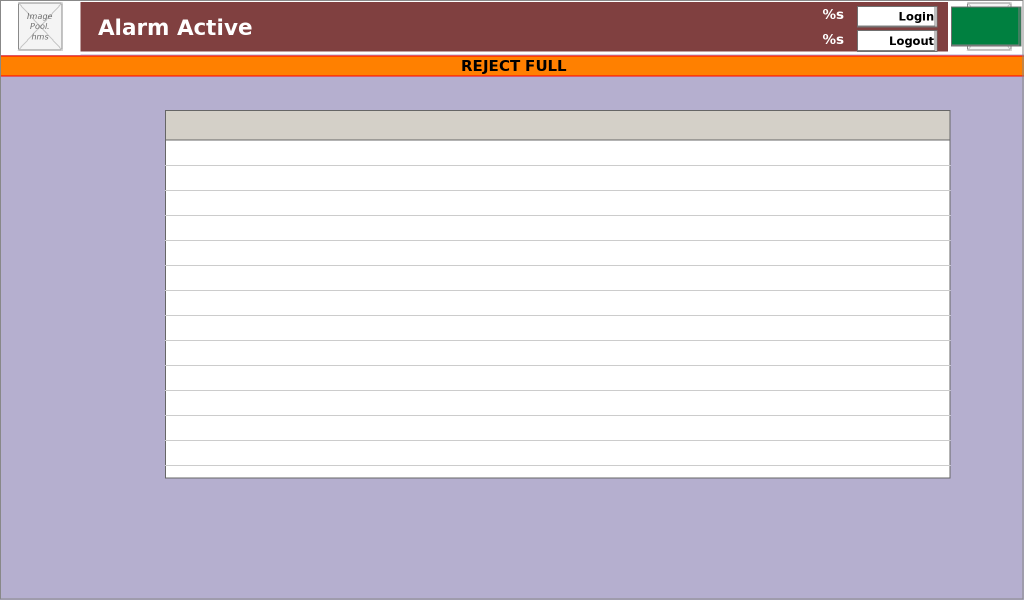
VISUALIZATION AlarmActive  // 1024x600
    Frame (0,-1 1024x55)
        shows Header()
    Label (95,15 250x25), "Alarm Active"
    Table (165,110 785x368), data array: Status_GVL.arAlarmActive
        p3854506369: Status_GVL.arAlarmActive[INDEX].Status
        p1892666644: Status_GVL.arAlarmActive[INDEX].ErrorID
        p338671338: Status_GVL.arAlarmActive[INDEX].ErrorMsg
        p2170511999: Status_GVL.arAlarmActive[INDEX].TimeStop
        p1755163831: Error Message
        p4092479075: Time Stop
END_VISUALIZATION

// ---- VISUs/Main/Alarm/Alarm.TcVIS
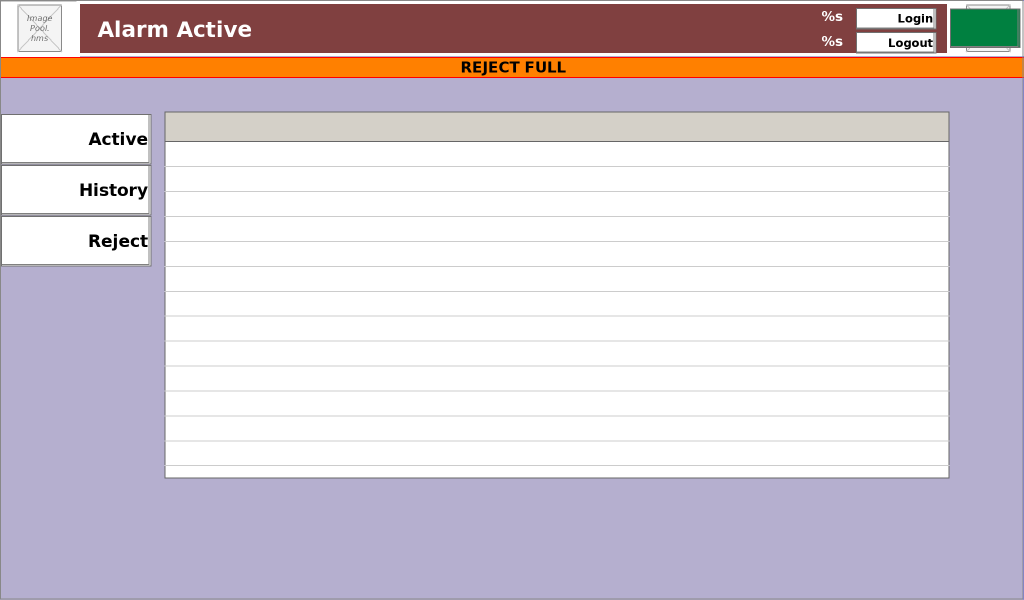
VISUALIZATION Alarm  // 1024x600
    Frame (0,2 1023x598)
        shows AlarmActive()
        shows AlarmHistory()
        shows RejectMsg()
        shows Test_Place1()
        shows Test_Place2()
        shows Test_Place3()
        shows Test_Place4()
    Button (1,114 150x50), "Active", image: VisuSymbols.Symbols.Database2
        OnMouseDown: FrameSelectionChange Selection=SelectedFrame=146e207b-fd78-4676-ba16-384fa245d7d2, GlobSel=AssignDir=MainPage.GenElemInst_1003, AssignType=Directly, SelType=Locally
    Button (1,165 150x50), "History", image: VisuSymbols.Symbols.Database2
        OnMouseDown: FrameSelectionChange Selection=SelectedFrame=146e207b-fd78-4676-ba16-384fa245d7d2, Selection=1, GlobSel=AssignDir=MainPage.GenElemInst_1003, AssignType=Directly, SelType=Locally
    Button (1,216 150x50), "Reject", image: VisuSymbols.Symbols.Database2
        OnMouseDown: FrameSelectionChange Selection=SelectedFrame=146e207b-fd78-4676-ba16-384fa245d7d2, Selection=2, GlobSel=AssignDir=MainPage.GenElemInst_1003, AssignType=Directly, SelType=Locally
END_VISUALIZATION

// ---- VISUs/Main/Alarm/PUDetail.TcVIS
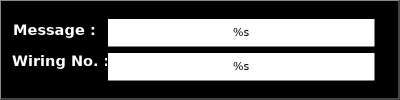
VISUALIZATION PUDetail  // 400x100
    Rectangle (0,0 400x100)
        OnMouseClick: CloseDialog Dialog=PUDetail, Result=None, NumpadKeypadSet=True
    Label (10,15 84x30), "Message :"
    Label (9,46 84x30), "Wiring No. :"
    Label (101,17 61x30)
    RoundedRectangle (107,18 268x29), "%s", tooltip "%s", text variable: HMI_GVL.sMessageError
        p4168582468: HMI_GVL.sMessageError
    RoundedRectangle (107,52 268x29), "%s", tooltip "%s", text variable: HMI_GVL.sWiringNo
        p4168582468: HMI_GVL.sWiringNo
END_VISUALIZATION

// ---- VISUs/Main/Header.TcVIS
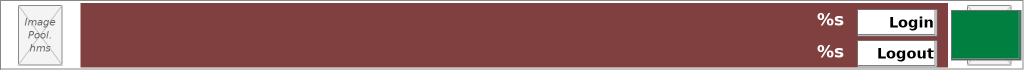
VISUALIZATION Header  // 1024x70
    Rectangle (77,0 947x70)
    Rectangle (535,39 312x25), "%s", text variable: visuelems.CurrentUserName
    Rectangle (948,0 79x70)
    Image (967,5 44x60), image: ImagePool.Logo
    Rectangle (0,72 1028x26), "MACHINE ERROR", invisible if: HMI_GVL.bMachineError
    Button (951,10 70x50), colour toggle: HMI_GVL.bMuteBuzzer, invisible if: HMI_GVL.bMachineError, image: VisuSymbols.Symbols.loudspeakerLoud
        toggle HMI_GVL.bMuteBuzzer
    Rectangle (1,1 79x70)
    Rectangle (0,72 1028x26), "REJECT FULL", invisible if: Status_GVL.RejectFull
    Image (18,5 44x60), image: ImagePool.hms
    Button (857,9 80x27), "Login", image: VisuSymbols.Symbols.User
        OnMouseDown: VisuUserMgmt Type=Login
    Rectangle (535,7 312x25), "%s", text variable: Status_GVL.strTimeEvent
    Button (857,40 80x27), "Logout", image: VisuSymbols.Symbols.User
        OnMouseDown: VisuUserMgmt Type=Logout
END_VISUALIZATION

// ---- VISUs/Main/Home.TcVIS
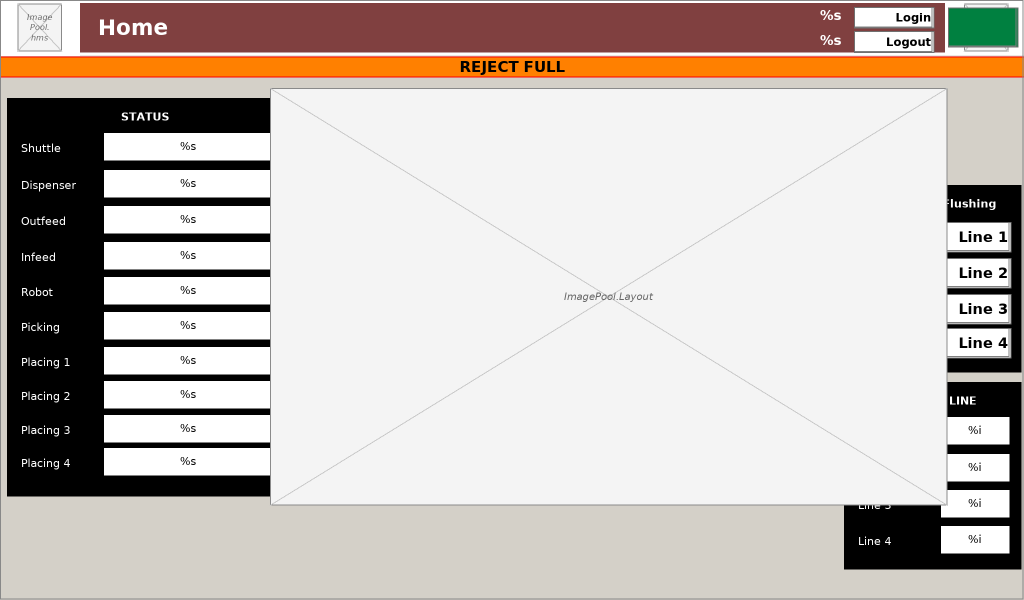
VISUALIZATION Home  // 1024x600
    RoundedRectangle (917,185 104x187)
    Frame (0,0 1021x55)
        shows Header()
    Label (95,15 214x25), "Home"
    RoundedRectangle (844,382 177x187)
    Label (869,381 125x40), "COUNTER LINE"
    Label (855,415 78x35), "Line 1"
    RoundedRectangle (940,416 70x29), "%i", text variable: HMI_GVL.arCountReal[1], input disabled if: Data_GVL.stStateMachineRobot.Running
        OnMouseClick: write the text variable via Default
    Label (855,452 78x35), "Line 2"
    RoundedRectangle (940,453 70x29), "%i", text variable: HMI_GVL.arCountReal[2], input disabled if: Data_GVL.stStateMachineRobot.Running
        OnMouseClick: write the text variable via Default
    Label (855,488 78x35), "Line 3"
    RoundedRectangle (940,489 70x29), "%i", text variable: HMI_GVL.arCountReal[3], input disabled if: Data_GVL.stStateMachineRobot.Running
        OnMouseClick: write the text variable via Default
    Label (855,524 78x35), "Line 4"
    RoundedRectangle (940,525 70x29), "%i", text variable: HMI_GVL.arCountReal[4], input disabled if: Data_GVL.stStateMachineRobot.Running
        OnMouseClick: write the text variable via Default
    Group (7,97 279x399)
        RoundedRectangle (0,1 279x398)
        Label (25,0 227x40), "STATUS"
        Label (11,34 78x35), "Shuttle"
        RoundedRectangle (96,35 170x29), "%s", text variable: InputOutput_GVL.Shuttle_stsMachine
        Label (11,71 78x35), "Dispenser"
        RoundedRectangle (96,72 170x29), "%s", text variable: InputOutput_GVL.Dispenser_stsMachine
        Label (11,107 78x35), "Outfeed"
        RoundedRectangle (96,108 170x29), "%s", text variable: InputOutput_GVL.Outfeed_stsMachine
        Label (11,143 78x35), "Infeed"
        RoundedRectangle (96,144 170x29), "%s", text variable: InputOutput_GVL.Infeed_stsMachine
        Label (11,178 78x35), "Robot"
        RoundedRectangle (96,179 170x29), "%s", text variable: Data_GVL.StateMachineRobot_stsMachine
        Label (11,213 78x35), "Picking"
        RoundedRectangle (96,214 170x29), "%s", text variable: Data_GVL.StateMachinePicking_stsMachine
        Label (11,248 78x35), "Placing 1"
        RoundedRectangle (96,249 170x29), "%s", text variable: Data_GVL.StateMachinePlacing1_stsMachine
        Label (11,282 78x35), "Placing 2"
        RoundedRectangle (96,283 170x29), "%s", text variable: Data_GVL.StateMachinePlacing2_stsMachine
        Label (11,316 78x35), "Placing 3"
        RoundedRectangle (96,317 170x29), "%s", text variable: Data_GVL.StateMachinePlacing3_stsMachine
        Label (11,349 78x35), "Placing 4"
        RoundedRectangle (96,350 170x29), "%s", text variable: Data_GVL.StateMachinePlacing4_stsMachine
    Button (930,222 81x30), "Line 1", image: VisuSymbols.Symbols.Rec
        tap HMI_GVL.Flush_Placing1
    Label (907,184 125x40), "Flushing"
    Button (930,258 81x30), "Line 2", image: VisuSymbols.Symbols.Rec
        tap HMI_GVL.Flush_Placing2
    Button (930,294 81x30), "Line 3", image: VisuSymbols.Symbols.Rec
        tap HMI_GVL.Flush_Placing3
    Button (930,328 81x30), "Line 4", image: VisuSymbols.Symbols.Rec
        tap HMI_GVL.Flush_Placing4
    Image (270,88 677x417), image: ImagePool.Layout
END_VISUALIZATION

// ---- VISUs/Main/MainPage.TcVIS
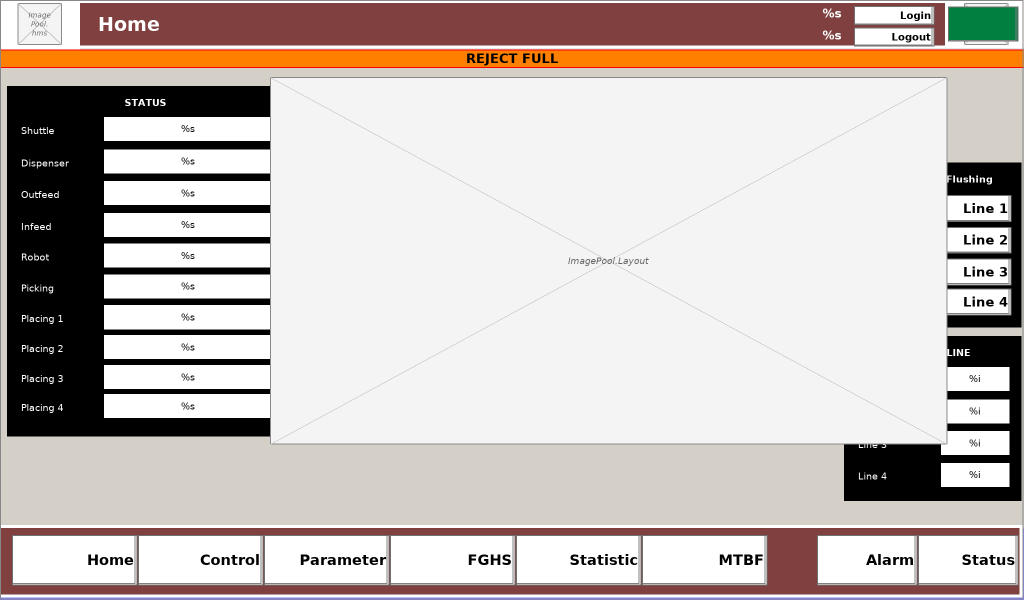
VISUALIZATION MainPage  // 1024x600
    Frame (0,0 1024x528)
        shows Home()
        shows Control()
        shows Parameter()
        shows FGHS()
        shows OEE()
        shows MTBF()
        shows Alarm()
        shows PLC_Status()
    Rectangle (-2,525 1024x72)
    Button (12,535 125x50), "Home", image: VisuSymbols.Symbols.Home
        OnMouseDown: FrameSelectionChange Selection=SelectedFrame=ea862550-edb1-43e7-b63a-bfe68bb940c3, GlobSel=AssignDir=MainPage.GenElemInst_1003, AssignType=Directly, SelType=Locally
    Button (138,535 125x50), "Control", image: VisuSymbols.Symbols.ControlPanel
        OnMouseDown: FrameSelectionChange Selection=SelectedFrame=ea862550-edb1-43e7-b63a-bfe68bb940c3, Selection=1, GlobSel=AssignType=Directly, SelType=Locally
    Button (817,535 100x50), "Alarm", image: VisuSymbols.Symbols.Caution
        OnMouseDown: FrameSelectionChange Selection=SelectedFrame=ea862550-edb1-43e7-b63a-bfe68bb940c3, Selection=6, GlobSel=AssignType=Directly, SelType=Locally
    Button (918,535 100x50), "Status", image: VisuSymbols.Symbols.Information
        OnMouseClick: FrameSelectionChange Selection=SelectedFrame=ea862550-edb1-43e7-b63a-bfe68bb940c3, Selection=7, GlobSel=AssignType=Directly, SelType=Locally
    Button (264,535 125x50), "Parameter", image: VisuSymbols.Symbols.TwoWheels
        OnMouseDown: FrameSelectionChange Selection=SelectedFrame=ea862550-edb1-43e7-b63a-bfe68bb940c3, Selection=2, GlobSel=AssignType=Directly, SelType=Locally
    Button (390,535 125x50), "FGHS", image: VisuSymbols.Symbols.Database
        OnMouseDown: FrameSelectionChange Selection=SelectedFrame=ea862550-edb1-43e7-b63a-bfe68bb940c3, Selection=3, GlobSel=AssignDir=MainPage.GenElemInst_1003, AssignType=Directly, SelType=Locally
    Button (516,535 125x50), "Statistic", image: VisuSymbols.Symbols.Diagram
        OnMouseDown: FrameSelectionChange Selection=SelectedFrame=ea862550-edb1-43e7-b63a-bfe68bb940c3, Selection=4, GlobSel=AssignDir=MainPage.GenElemInst_1003, AssignType=Directly, SelType=Locally
    Button (642,535 125x50), "MTBF", image: VisuSymbols.Symbols.Chart
        OnMouseDown: FrameSelectionChange Selection=SelectedFrame=ea862550-edb1-43e7-b63a-bfe68bb940c3, Selection=5, GlobSel=AssignDir=MainPage.GenElemInst_1003, AssignType=Directly, SelType=Locally
END_VISUALIZATION

// ---- VISUs/Main/Parameter.TcVIS
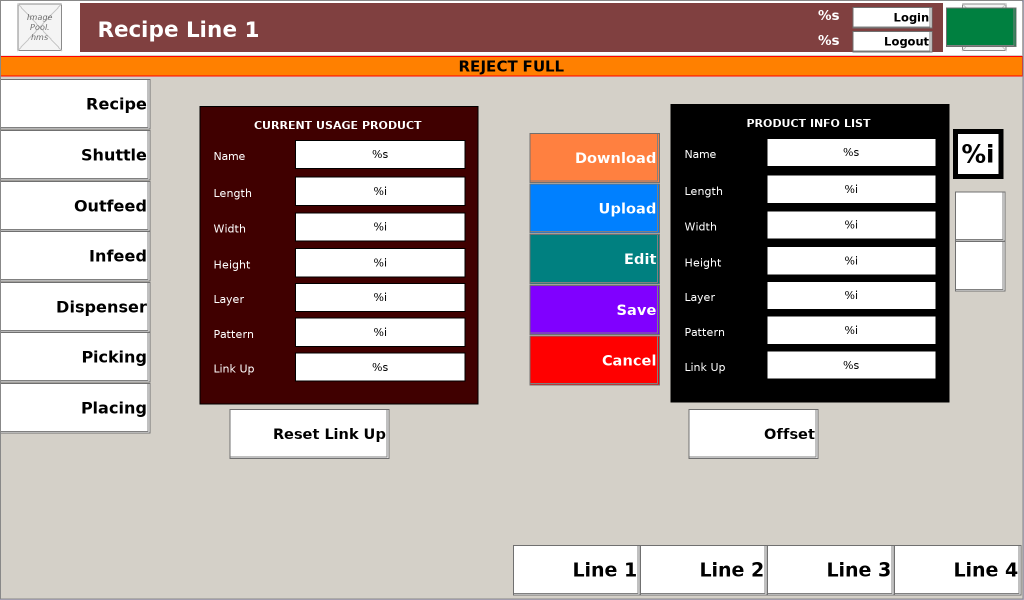
VISUALIZATION Parameter  // 1024x600
    Frame (0,0 1023x598)
        shows MRecipe()
        shows MShuttle()
        shows MOutfeed()
        shows MInfeed()
        shows MDispenser()
        shows MPicking()
        shows MPlacing()
        shows Test_Infeed()
        shows Test_Picking()
    Button (0,79 150x50), "Recipe", image: VisuSymbols.Symbols.Database2
        OnMouseDown: FrameSelectionChange Selection=SelectedFrame=5d0adf46-92b2-4ae0-bcf1-a330fcf05353, GlobSel=AssignDir=MainPage.GenElemInst_1003, AssignType=Directly, SelType=Locally
    Button (0,130 150x50), "Shuttle", image: VisuSymbols.Symbols.Database2
        OnMouseDown: FrameSelectionChange Selection=SelectedFrame=5d0adf46-92b2-4ae0-bcf1-a330fcf05353, Selection=1, GlobSel=AssignDir=MainPage.GenElemInst_1003, AssignType=Directly, SelType=Locally
    Button (0,181 150x50), "Outfeed", image: VisuSymbols.Symbols.Database2
        OnMouseDown: FrameSelectionChange Selection=SelectedFrame=5d0adf46-92b2-4ae0-bcf1-a330fcf05353, Selection=2, GlobSel=AssignDir=MainPage.GenElemInst_1003, AssignType=Directly, SelType=Locally
    Button (0,231 150x50), "Infeed", image: VisuSymbols.Symbols.Database2
        OnMouseDown: FrameSelectionChange Selection=SelectedFrame=5d0adf46-92b2-4ae0-bcf1-a330fcf05353, Selection=3, GlobSel=AssignDir=MainPage.GenElemInst_1003, AssignType=Directly, SelType=Locally
    Button (0,282 150x50), "Dispenser", image: VisuSymbols.Symbols.Database2
        OnMouseDown: FrameSelectionChange Selection=SelectedFrame=5d0adf46-92b2-4ae0-bcf1-a330fcf05353, Selection=4, GlobSel=AssignDir=MainPage.GenElemInst_1003, AssignType=Directly, SelType=Locally
    Button (0,332 150x50), "Picking", image: VisuSymbols.Symbols.Database2
        OnMouseDown: FrameSelectionChange Selection=SelectedFrame=5d0adf46-92b2-4ae0-bcf1-a330fcf05353, Selection=5, GlobSel=AssignDir=MainPage.GenElemInst_1003, AssignType=Directly, SelType=Locally
    Button (0,383 150x50), "Placing", image: VisuSymbols.Symbols.Database2
        OnMouseDown: FrameSelectionChange Selection=SelectedFrame=5d0adf46-92b2-4ae0-bcf1-a330fcf05353, Selection=6, GlobSel=AssignDir=MainPage.GenElemInst_1003, AssignType=Directly, SelType=Locally
END_VISUALIZATION

// ---- VISUs/Main/PLC_Status.TcVIS
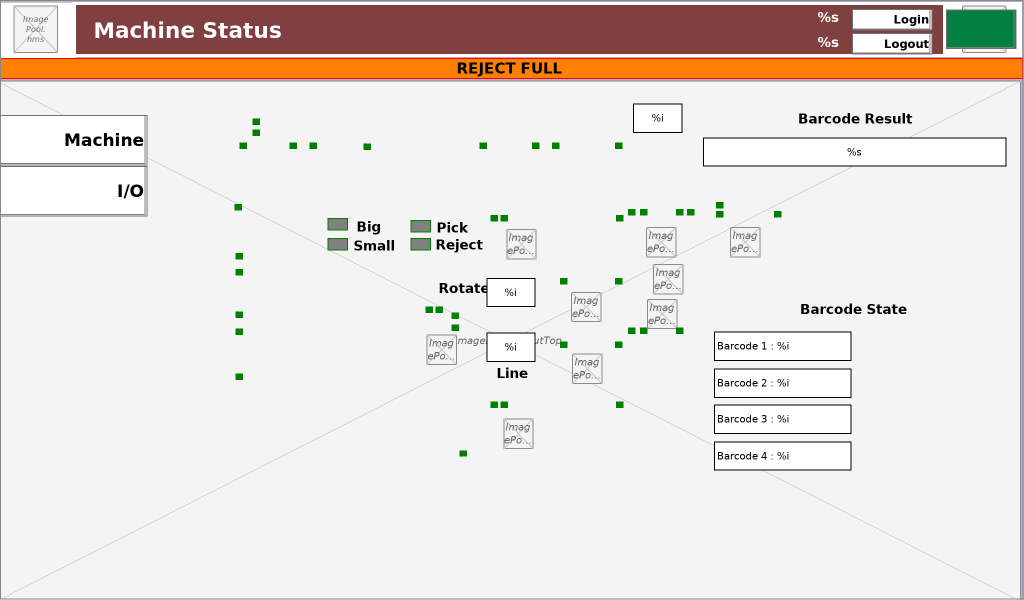
VISUALIZATION PLC_Status  // 1024x600
    Frame (-4,3 1023x598)
        shows SeqStatus()
        shows IO_Status()
        shows Test_Shuttle()
        shows Test_Place1()
        shows Test_Place2()
        shows Test_Place3()
        shows Test_Place4()
    Button (-3,115 150x50), "Machine", image: VisuSymbols.Symbols.Database2
        OnMouseDown: FrameSelectionChange Selection=SelectedFrame=eb142f5b-097c-4dbf-af2f-09085337604c, GlobSel=AssignDir=MainPage.GenElemInst_1003, AssignType=Directly, SelType=Locally
    Button (-3,166 150x50), "I/O", image: VisuSymbols.Symbols.Database2
        OnMouseDown: FrameSelectionChange Selection=SelectedFrame=eb142f5b-097c-4dbf-af2f-09085337604c, Selection=1, GlobSel=AssignDir=MainPage.GenElemInst_1003, AssignType=Directly, SelType=Locally
END_VISUALIZATION

// ---- VISUs/Main/PUSeq.TcVIS
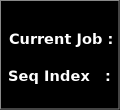
VISUALIZATION PUSeq  // 120x110
    Rectangle (0,0 371x118)
        OnMouseDown: CloseDialog Dialog=PUSeq, Result=None, NumpadKeypadSet=True
    Label (6,24 114x30), "Current Job :"
    Label (126,23 61x30)
    RoundedRectangle (121,24 235x29), "%s", tooltip "%s", text variable: HMI_GVL.sCurrentJob
        p4168582468: HMI_GVL.sCurrentJob
    RoundedRectangle (121,61 235x29), "%i", tooltip "%i", text variable: HMI_GVL.iSeqIndex
        p4168582468: HMI_GVL.iSeqIndex
    Label (5,61 121x30), "Seq Index :"
END_VISUALIZATION

// ---- VISUs/Main/StateMachine.TcVIS
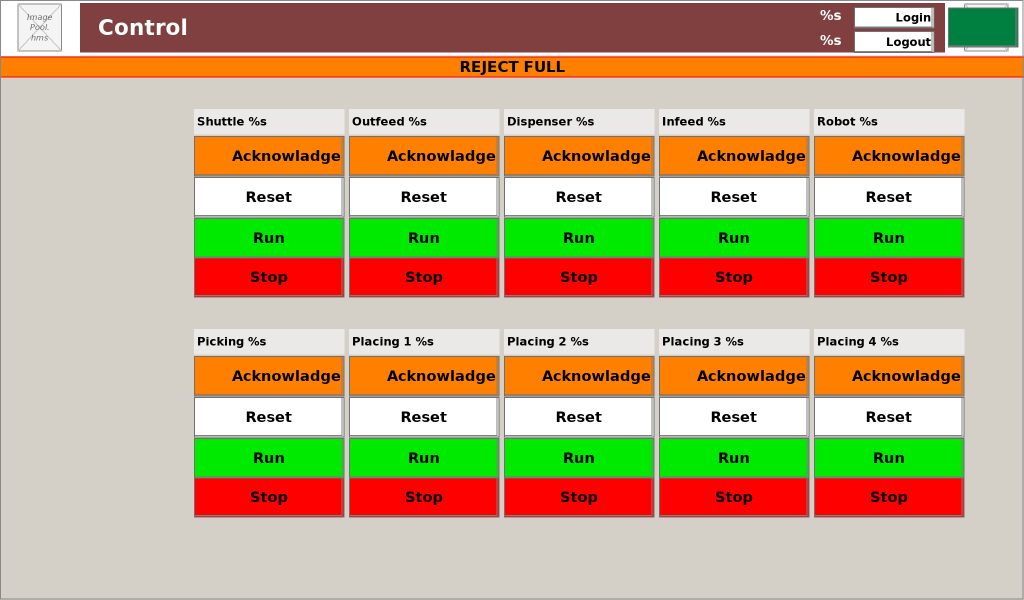
VISUALIZATION StateMachine  // 1024x600
    Frame (0,0 1021x55)
        shows Header()
    Group (194,109 150x188)
        Button (0,27 150x40), "Acknowladge", image: VisuSymbols.Symbols.OK
            tap HMI_GVL.bAcknowledgeButtonShuttle
        Button (0,68 150x40), "Reset", image: VisuSymbols.Symbols.Rec
            tap HMI_GVL.bResetButtonShuttle
        Button (0,148 150x40), "Stop", image: VisuSymbols.Symbols.Stop
            tap HMI_GVL.bStopButtonShuttle
        Button (0,109 150x40), "Run", image: VisuSymbols.Symbols.Play
            tap HMI_GVL.bStartButtonShuttle
        Rectangle (0,0 150x25), "Shuttle %s", text variable: InputOutput_GVL.Shuttle_stsMachine
    Button (349,136 150x40), "Acknowladge", image: VisuSymbols.Symbols.OK
        tap HMI_GVL.bAcknowledgeButtonOutfeed
    Button (349,177 150x40), "Reset", image: VisuSymbols.Symbols.Rec
        tap HMI_GVL.bResetButtonOutfeed
    Button (349,257 150x40), "Stop", image: VisuSymbols.Symbols.Stop
        tap HMI_GVL.bStopButtonOutfeed
    Button (349,218 150x40), "Run", image: VisuSymbols.Symbols.Play
        tap HMI_GVL.bStartButtonOutfeed
    Rectangle (349,109 150x25), "Outfeed %s", text variable: InputOutput_GVL.Outfeed_stsMachine
    Button (504,136 150x40), "Acknowladge", image: VisuSymbols.Symbols.OK
        tap HMI_GVL.bAcknowledgeButtonDispenser
    Button (504,177 150x40), "Reset", image: VisuSymbols.Symbols.Rec
        tap HMI_GVL.bResetButtonDispenser
    Button (504,257 150x40), "Stop", image: VisuSymbols.Symbols.Stop
        tap HMI_GVL.bStopButtonDispenser
    Button (504,218 150x40), "Run", image: VisuSymbols.Symbols.Play
        tap HMI_GVL.bStartButtonDispenser
    Rectangle (504,109 150x25), "Dispenser %s", text variable: InputOutput_GVL.Dispenser_stsMachine
    Group (659,109 150x188)
        Button (0,27 150x40), "Acknowladge", image: VisuSymbols.Symbols.OK
            tap HMI_GVL.bAcknowledgeButtonInfeed
        Button (0,68 150x40), "Reset", image: VisuSymbols.Symbols.Rec
            tap HMI_GVL.bResetButtonInfeed
        Button (0,148 150x40), "Stop", image: VisuSymbols.Symbols.Stop
            tap HMI_GVL.bStopButtonInfeed
        Button (0,109 150x40), "Run", image: VisuSymbols.Symbols.Play
            tap HMI_GVL.bStartButtonInfeed
        Rectangle (0,0 150x25), "Infeed %s", text variable: InputOutput_GVL.Infeed_stsMachine
    Group (814,109 150x188)
        Button (0,27 150x40), "Acknowladge", image: VisuSymbols.Symbols.OK
            tap HMI_GVL.bAcknowledgeButtonRobot
        Button (0,68 150x40), "Reset", image: VisuSymbols.Symbols.Rec
            tap HMI_GVL.bResetButtonRobot
        Button (0,148 150x40), "Stop", image: VisuSymbols.Symbols.Stop
            tap HMI_GVL.bStopButtonRobot
        Button (0,109 150x40), "Run", image: VisuSymbols.Symbols.Play
            tap HMI_GVL.bStartButtonRobot
        Rectangle (0,0 150x25), "Robot %s", text variable: Data_GVL.StateMachineRobot_stsMachine
    Button (194,356 150x40), "Acknowladge", image: VisuSymbols.Symbols.OK
        tap HMI_GVL.bAcknowledgeButtonPicking
    Button (194,397 150x40), "Reset", image: VisuSymbols.Symbols.Rec
        tap HMI_GVL.bResetButtonPicking
    Button (194,477 150x40), "Stop", image: VisuSymbols.Symbols.Stop
        tap HMI_GVL.bStopButtonPicking
    Button (194,438 150x40), "Run", image: VisuSymbols.Symbols.Play
        tap HMI_GVL.bStartButtonPicking
    Rectangle (194,329 150x25), "Picking %s", text variable: Data_GVL.StateMachinePicking_stsMachine
    Button (349,356 150x40), "Acknowladge", image: VisuSymbols.Symbols.OK
        tap HMI_GVL.bAcknowledgeButtonPlacing1
    Button (349,397 150x40), "Reset", image: VisuSymbols.Symbols.Rec
        tap HMI_GVL.bResetButtonPlacing1
    Button (349,477 150x40), "Stop", image: VisuSymbols.Symbols.Stop
        tap HMI_GVL.bStopButtonPlacing1
    Button (349,438 150x40), "Run", image: VisuSymbols.Symbols.Play
        tap HMI_GVL.bStartButtonPlacing1
    Rectangle (349,329 150x25), "Placing 1 %s", text variable: Data_GVL.StateMachinePlacing1_stsMachine
    Button (504,356 150x40), "Acknowladge", image: VisuSymbols.Symbols.OK
        tap HMI_GVL.bAcknowledgeButtonPlacing2
    Button (504,397 150x40), "Reset", image: VisuSymbols.Symbols.Rec
        tap HMI_GVL.bResetButtonPlacing2
    Button (504,477 150x40), "Stop", image: VisuSymbols.Symbols.Stop
        tap HMI_GVL.bStopButtonPlacing2
    Button (504,438 150x40), "Run", image: VisuSymbols.Symbols.Play
        tap HMI_GVL.bStartButtonPlacing2
    Rectangle (504,329 150x25), "Placing 2 %s", text variable: Data_GVL.StateMachinePlacing2_stsMachine
    Button (659,356 150x40), "Acknowladge", image: VisuSymbols.Symbols.OK
        tap HMI_GVL.bAcknowledgeButtonPlacing3
    Button (659,397 150x40), "Reset", image: VisuSymbols.Symbols.Rec
        tap HMI_GVL.bResetButtonPlacing3
    Button (659,477 150x40), "Stop", image: VisuSymbols.Symbols.Stop
        tap HMI_GVL.bStopButtonPlacing3
    Button (659,438 150x40), "Run", image: VisuSymbols.Symbols.Play
        tap HMI_GVL.bStartButtonPlacing3
    Rectangle (659,329 150x25), "Placing 3 %s", text variable: Data_GVL.StateMachinePlacing3_stsMachine
    Button (814,356 150x40), "Acknowladge", image: VisuSymbols.Symbols.OK
        tap HMI_GVL.bAcknowledgeButtonPlacing4
    Button (814,397 150x40), "Reset", image: VisuSymbols.Symbols.Rec
        tap HMI_GVL.bResetButtonPlacing4
    Button (814,477 150x40), "Stop", image: VisuSymbols.Symbols.Stop
        tap HMI_GVL.bStopButtonPlacing4
    Button (814,438 150x40), "Run", image: VisuSymbols.Symbols.Play
        tap HMI_GVL.bStartButtonPlacing4
    Rectangle (814,329 150x25), "Placing 4 %s", text variable: Data_GVL.StateMachinePlacing4_stsMachine
    Label (95,15 214x25), "Control"
END_VISUALIZATION

// ---- VISUs/MTBF/MTBF.TcVIS
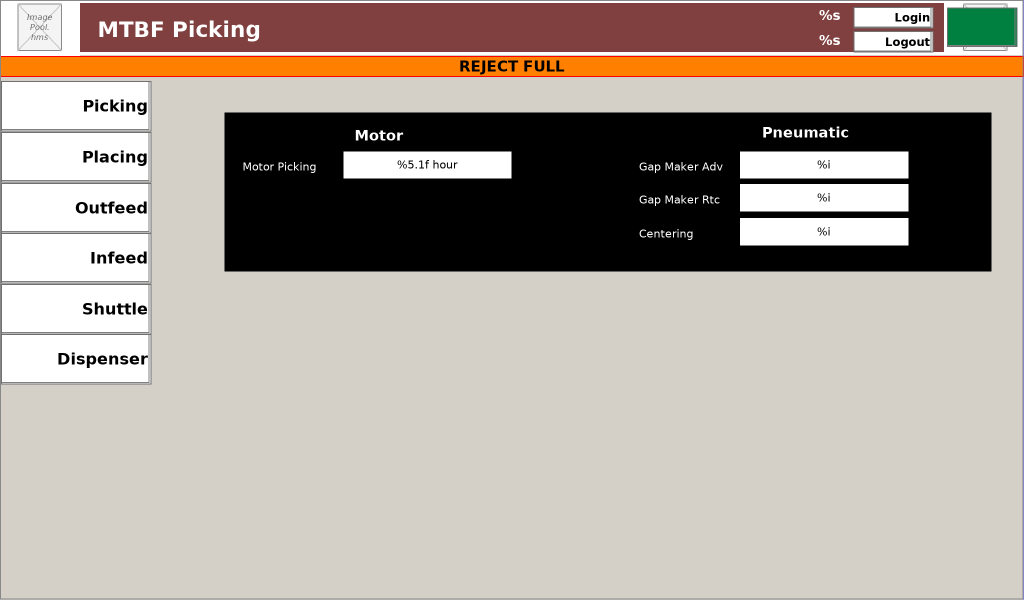
VISUALIZATION MTBF  // 1024x600
    Frame (0,2 1023x598)
        shows MTBF_Picking()
        shows MTBF_Placing()
        shows MTBF_Outfeed()
        shows MTBF_Infeed()
        shows MTBF_Shuttle()
        shows MTBF_Dispenser()
        shows Test_Place4()
        shows Test_Infeed()
        shows Test_Picking()
    Button (1,81 150x50), "Picking", image: VisuSymbols.Symbols.Database2
        OnMouseDown: FrameSelectionChange Selection=SelectedFrame=146e207b-fd78-4676-ba16-384fa245d7d2, GlobSel=AssignDir=MainPage.GenElemInst_1003, AssignType=Directly, SelType=Locally
    Button (1,132 150x50), "Placing", image: VisuSymbols.Symbols.Database2
        OnMouseDown: FrameSelectionChange Selection=SelectedFrame=146e207b-fd78-4676-ba16-384fa245d7d2, Selection=1, GlobSel=AssignDir=MainPage.GenElemInst_1003, AssignType=Directly, SelType=Locally
    Button (1,183 150x50), "Outfeed", image: VisuSymbols.Symbols.Database2
        OnMouseDown: FrameSelectionChange Selection=SelectedFrame=146e207b-fd78-4676-ba16-384fa245d7d2, Selection=2, GlobSel=AssignDir=MainPage.GenElemInst_1003, AssignType=Directly, SelType=Locally
    Button (1,233 150x50), "Infeed", image: VisuSymbols.Symbols.Database2
        OnMouseDown: FrameSelectionChange Selection=SelectedFrame=146e207b-fd78-4676-ba16-384fa245d7d2, Selection=3, GlobSel=AssignDir=MainPage.GenElemInst_1003, AssignType=Directly, SelType=Locally
    Button (1,284 150x50), "Shuttle", image: VisuSymbols.Symbols.Database2
        OnMouseDown: FrameSelectionChange Selection=SelectedFrame=146e207b-fd78-4676-ba16-384fa245d7d2, Selection=4, GlobSel=AssignDir=MainPage.GenElemInst_1003, AssignType=Directly, SelType=Locally
    Button (1,334 150x50), "Dispenser", image: VisuSymbols.Symbols.Database2
        OnMouseDown: FrameSelectionChange Selection=SelectedFrame=146e207b-fd78-4676-ba16-384fa245d7d2, Selection=5, GlobSel=AssignDir=MainPage.GenElemInst_1003, AssignType=Directly, SelType=Locally
END_VISUALIZATION

// ---- VISUs/MTBF/MTBF_Picking.TcVIS
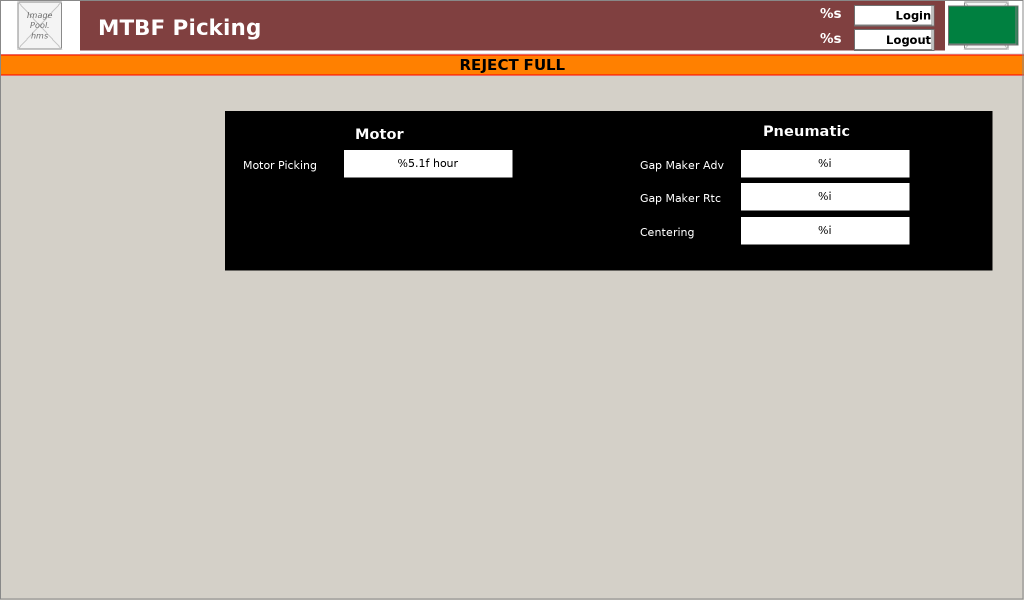
VISUALIZATION MTBF_Picking  // 1024x600
    Frame (0,-2 1021x55)
        shows Header()
    Label (95,15 250x25), "MTBF Picking"
    RoundedRectangle (225,111 767x159)
    Label (243,114 273x40), "Motor"
    Label (240,148 103x35), "Motor Picking"
    RoundedRectangle (343,149 170x29), "%5.1f hour", text variable: Status_GVL.stMotor_Picking.RunningHours
    Label (637,148 104x35), "Gap Maker Adv"
    RoundedRectangle (740,149 170x29), "%i", text variable: Status_GVL.stPneu_GapMaker.CyclePneuAdv
    Label (670,111 273x40), "Pneumatic"
    Label (637,181 104x35), "Gap Maker Rtc"
    RoundedRectangle (740,182 170x29), "%i", text variable: Status_GVL.stPneu_GapMaker.CyclePneuRtc
    Label (637,215 104x35), "Centering"
    RoundedRectangle (740,216 170x29), "%i", text variable: Status_GVL.stPneu_Centering.CyclePneu
END_VISUALIZATION

// ---- VISUs/MTBF/MTBF_Placing.TcVIS
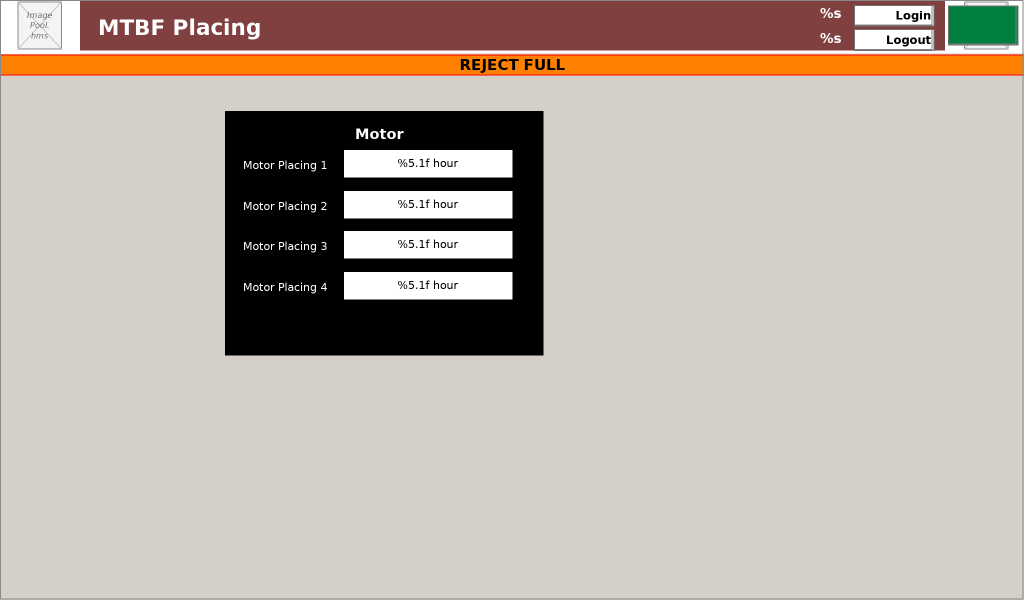
VISUALIZATION MTBF_Placing  // 1024x600
    Frame (0,-2 1021x55)
        shows Header()
    Label (95,15 250x25), "MTBF Placing"
    RoundedRectangle (225,111 318x244)
    Label (243,114 273x40), "Motor"
    Label (240,148 103x35), "Motor Placing 1"
    RoundedRectangle (343,149 170x29), "%5.1f hour", text variable: Status_GVL.stMotor_Placing1.RunningHours
    Label (240,189 103x35), "Motor Placing 2"
    RoundedRectangle (343,190 170x29), "%5.1f hour", text variable: Status_GVL.stMotor_Placing2.RunningHours
    Label (240,229 103x35), "Motor Placing 3"
    RoundedRectangle (343,230 170x29), "%5.1f hour", text variable: Status_GVL.stMotor_Placing3.RunningHours
    Label (240,270 103x35), "Motor Placing 4"
    RoundedRectangle (343,271 170x29), "%5.1f hour", text variable: Status_GVL.stMotor_Placing4.RunningHours
END_VISUALIZATION

// ---- VISUs/MTBF/MTBF_Outfeed.TcVIS
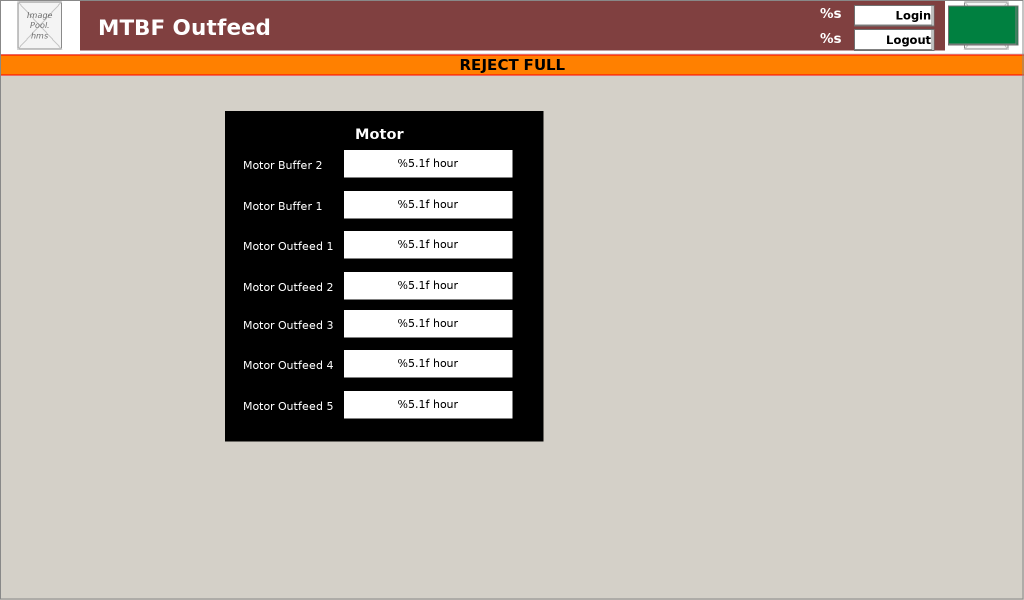
VISUALIZATION MTBF_Outfeed  // 1024x600
    Frame (0,-2 1021x55)
        shows Header()
    Label (95,15 250x25), "MTBF Outfeed"
    RoundedRectangle (225,111 318x330)
    Label (243,114 273x40), "Motor"
    Label (240,148 103x35), "Motor Buffer 2"
    RoundedRectangle (343,149 170x29), "%5.1f hour", text variable: InputOutput_GVL.MTBF_Motor[1]
    Label (240,189 103x35), "Motor Buffer 1"
    RoundedRectangle (343,190 170x29), "%5.1f hour", text variable: InputOutput_GVL.MTBF_Motor[2]
    Label (240,229 103x35), "Motor Outfeed 1"
    RoundedRectangle (343,230 170x29), "%5.1f hour", text variable: InputOutput_GVL.MTBF_Motor[3]
    Label (240,270 103x35), "Motor Outfeed 2"
    RoundedRectangle (343,271 170x29), "%5.1f hour", text variable: InputOutput_GVL.MTBF_Motor[4]
    Label (240,308 103x35), "Motor Outfeed 3"
    RoundedRectangle (343,309 170x29), "%5.1f hour", text variable: InputOutput_GVL.MTBF_Motor[5]
    Label (240,348 103x35), "Motor Outfeed 4"
    RoundedRectangle (343,349 170x29), "%5.1f hour", text variable: InputOutput_GVL.MTBF_Motor[6]
    Label (240,389 103x35), "Motor Outfeed 5"
    RoundedRectangle (343,390 170x29), "%5.1f hour", text variable: InputOutput_GVL.MTBF_Motor[7]
END_VISUALIZATION

// ---- VISUs/MTBF/MTBF_Infeed.TcVIS
